ABB RobotStudio station: Universo_updated.rspag

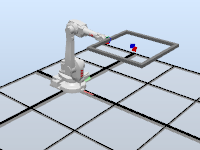
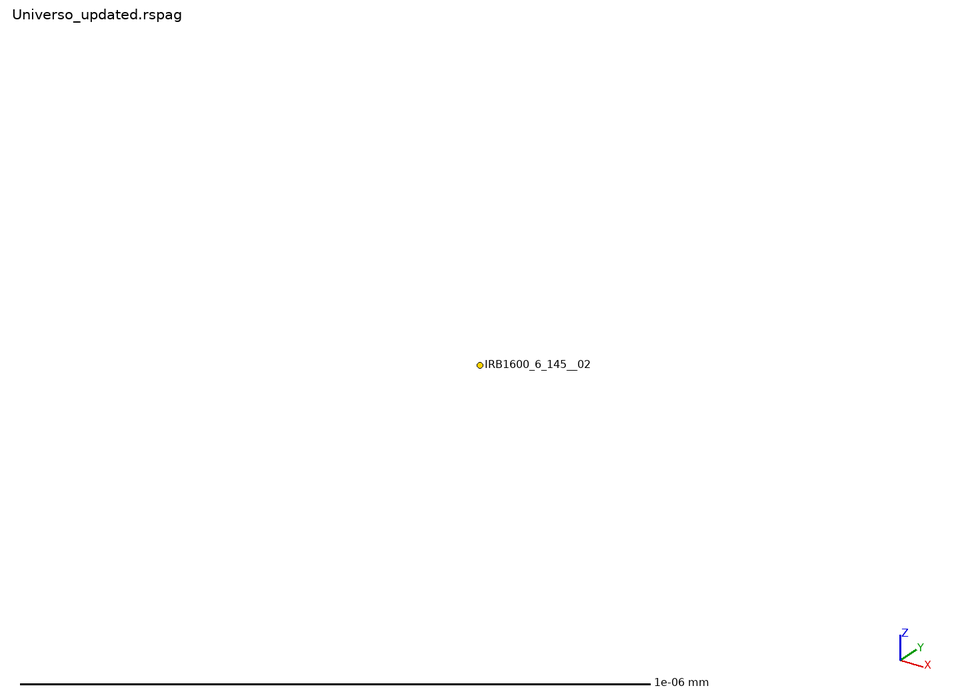
[picture v1: parts stored in the station drawn from their meshes, with robot base, taught points and paths (robot models come from the ABB library and are not in the file)]
--- station ---
Station Solution1 (saved by RobotStudio 22.1.9826.0)
Controller IRB1600_6_145
  mechanical unit ROB_1: IRB1600_6_145__02, 6 joints, base frame (0, 0, 0) mm
Layout (positions relative to the parent item):
  - IRB1600_6_145__02 [mechanism, from Robots\IRB1600_6_145_G_02.rslib] at (0, 0, 0) mm; joint values [-0.0012, -0.0048, 0.0813, -0.0158, -0.0765, 0.0158] (rad or m)
  - flange_connector [part, from Tools\IsoPlate_small_Binzel.rslib] at (809.87, -0.9, 1140.62) mm, rotated rx 0 ry 90 rz 0 deg
  - plane [part] at (1319.2, 1.57, 1145.26) mm, rotated rx 180 ry 0 rz 180 deg, size 1000 x 1000 x 50 mm
  - Frame_1 [frame]
  - Frame_2 [frame] at (-23.65, -1.83, 250.36) mm
Attachment: flange_connector is attached to IRB1600_6_145__02 / Link6
Attachment: plane is attached to flange_connector
Attachment: Workobject_2 is attached to IRB1600_6_145__02 / Link1
Targets, tools, work objects and paths stored in the station and not in the controller backup, written as RAPID:
! task T_ROB1
MODULE Module1
  LOCAL PERS wobjdata egm_wobj:=[FALSE,TRUE,"",[[0,0,0],[1,0,0,0]],[[0,0,0],[1,0,0,0]]];
  PROC EGM_CARTESIAN_MOVE()
    WaitTime 2;
  ENDPROC
ENDMODULE


--- Backups/IRB1600_6_145/RAPID/TASK1/PROGMOD/CalibData.mod ---
MODULE CalibData
    TASK PERS tooldata Tooldata_3:=[TRUE,[[-23.481,11.123,47.179],[0.707106781,0,0.707106781,0]],[1,[0,0,1],[1,0,0,0],0,0,0]];
    TASK PERS tooldata Tooldata_8:=[TRUE,[[35.292999999,18.761,1471.373000001],[0.707106781,0,-0.707106781,0]],[1,[0,0,1],[1,0,0,0],0,0,0]];
    TASK PERS tooldata Tooldata_4:=[TRUE,[[0,0,0],[1,0,0,0]],[1,[0,0,1],[1,0,0,0],0,0,0]];
    TASK PERS tooldata Tooldata_5:=[TRUE,[[0,0,0],[1,0,0,0]],[1,[0,0,1],[1,0,0,0],0,0,0]];
    TASK PERS tooldata Tooldata_6:=[TRUE,[[0,0,0],[1,0,0,0]],[1,[0,0,1],[1,0,0,0],0,0,0]];
    TASK PERS tooldata Tooldata_7:=[TRUE,[[-23.772999698,2.161000196,740.120999999],[0.707106781,0,-0.707106781,0]],[1,[0,0,1],[1,0,0,0],0,0,0]];
    TASK PERS wobjdata Workobject_2:=[FALSE,TRUE,"ROB_1",[[-55.133477186,-6.202200727,258.13059393],[1,0,0,0]],[[0,0,0],[1,0,0,0]]];
    TASK PERS tooldata Tooldata_9:=[TRUE,[[20.616002648,0.899999913,497.265999882],[0.707106781,-0.000000002,-0.707106781,0]],[1,[0,0,1],[1,0,0,0],0,0,0]];
    TASK PERS wobjdata Wobj_joint1:=[TRUE,FALSE,"ROB_1",[[639.116,-613.962,-938.233],[1,0,0,0]],[[0,0,0],[1,0,0,0]]];
ENDMODULE

--- Backups/IRB1600_6_145/RAPID/TASK1/PROGMOD/Module1.mod ---
MODULE Module1

     VAR robtarget position;
     VAR robtarget starting_position;
     VAR jointtarget joints;
     VAR speeddata velocity;
    TASK PERS wobjdata wobj:=[FALSE,FALSE,"ROB_1",[[639.116,-22.796,-980.437],[1,0,0,0]],[[0,0,0],[1,0,0,0]]];

    PROC main()

starting_position := CRobT(\TaskName:="T_ROB1" \Tool:=Tooldata_9 \WObj:=Workobject_2);
move 223,-627.8,7,20.4,0,0.9;
move 222,-628.9,7,20.4,15,1;
move 222,-630.1,6.9,20.4,15,1;
move 221,-631.2,6.9,20,15,1;
move 220,-632.5,6.9,20,15,1.1;
move 219,-633.7,6.8,19.6,15,1.1;
move 218,-635,6.8,19.6,15,1.2;
move 217,-636.4,6.8,19.2,15,1.2;
move 216,-637.8,6.8,19.2,15,1.2;
move 214,-639.3,6.8,18.8,15,1.3;
move 213,-640.8,6.8,18.8,15,1.3;
move 211,-642.4,6.8,18.4,14.9,1.4;
move 210,-644,6.8,18.4,14.9,1.4;
move 208,-645.6,6.7,18,14.9,1.5;
move 207,-647.3,6.7,18,14.9,1.5;
move 205,-649,6.7,17.6,14.9,1.6;
move 204,-650.7,6.7,17.6,14.9,1.6;
move 202,-652.4,6.6,17.2,14.9,1.7;
move 201,-654.1,6.6,16.8,14.8,1.7;
move 199,-655.8,6.6,16.8,14.8,1.8;
move 198,-657.5,6.6,16.8,14.8,1.9;
move 196,-659.2,6.6,16.4,14.8,1.9;
move 194,-660.8,6.6,16.4,14.8,2;
move 193,-662.4,6.6,16,14.7,2;
move 191,-664,6.6,15.6,14.7,2.1;
move 190,-665.6,6.5,15.6,14.7,2.2;
move 188,-667.2,6.5,15.2,14.7,2.2;
move 186,-668.7,6.5,15.2,14.6,2.3;
move 185,-670.2,6.5,14.8,14.6,2.4;
move 183,-671.6,6.5,14.8,14.6,2.4;
move 181,-673,6.5,14.4,14.5,2.5;
move 179,-674.3,6.5,14,14.5,2.6;
move 177,-675.5,6.4,14,14.5,2.7;
move 176,-676.7,6.4,13.6,14.5,2.7;
move 174,-677.8,6.4,13.2,14.4,2.8;
move 172,-678.8,6.4,13.2,14.4,2.9;
move 170,-679.8,6.4,12.8,14.3,2.9;
move 169,-680.7,6.4,12.8,14.3,3;
move 167,-681.6,6.4,12.4,14.3,3.1;
move 165,-682.4,6.4,12.4,14.2,3.2;
move 164,-683.2,6.4,12,14.2,3.3;
move 162,-683.9,6.4,11.6,14.2,3.3;
move 160,-684.7,6.3,11.6,14.1,3.4;
move 159,-685.4,6.3,11.2,14.1,3.5;
move 157,-686.1,6.3,11.2,14,3.6;
move 155,-686.7,6.3,10.8,14,3.6;
move 154,-687.4,6.3,10.8,13.9,3.7;
move 152,-688.1,6.3,10.4,13.9,3.8;
move 150,-688.8,6.2,10,13.8,3.9;
move 149,-689.5,6.2,10,13.8,4;
move 147,-690.2,6.2,9.6,13.7,4;
move 145,-690.9,6.2,9.6,13.7,4.1;
move 144,-691.6,6.2,9.2,13.6,4.2;
move 142,-692.3,6.2,9.2,13.6,4.3;
move 141,-693,6.1,8.8,13.5,4.3;
move 139,-693.6,6.1,8.8,13.5,4.4;
move 138,-694.3,6.1,8.4,13.4,4.5;
move 136,-694.9,6.1,8.4,13.4,4.6;
move 135,-695.5,6,8,13.3,4.6;
move 134,-696.1,6,8,13.3,4.7;
move 132,-696.6,6,7.6,13.2,4.8;
move 131,-697.1,5.9,7.6,13.1,4.9;
move 129,-697.6,5.9,7.2,13.1,4.9;
move 128,-698,5.9,7.2,13,5;
move 126,-698.4,5.8,6.8,12.9,5.1;
move 125,-698.8,5.8,6.8,12.9,5.1;
move 123,-699.2,5.8,6.4,12.8,5.2;
move 122,-699.5,5.7,6.4,12.8,5.3;
move 121,-699.8,5.7,6,12.7,5.4;
move 119,-700.1,5.6,6,12.6,5.4;
move 118,-700.3,5.6,5.6,12.6,5.5;
move 117,-700.6,5.6,5.6,12.5,5.6;
move 116,-700.8,5.5,5.6,12.4,5.6;
move 114,-701.1,5.5,5.2,12.3,5.7;
move 113,-701.3,5.4,5.2,12.3,5.8;
move 112,-701.6,5.4,4.8,12.2,5.8;
move 111,-701.8,5.3,4.8,12.1,5.9;
move 110,-702.1,5.2,4.8,12.1,6;
move 109,-702.4,5.2,4.4,12,6;
move 108,-702.7,5.1,4.4,11.9,6.1;
move 106,-703,5.1,4.4,11.8,6.2;
move 105,-703.3,5,4,11.7,6.2;
move 104,-703.7,4.9,4,11.7,6.3;
move 103,-704,4.9,3.6,11.6,6.3;
move 102,-704.4,4.8,3.6,11.5,6.4;
move 101,-704.8,4.7,3.6,11.4,6.5;
move 100,-705.2,4.7,3.2,11.3,6.5;
move 99,-705.6,4.6,3.2,11.3,6.6;
move 98,-706,4.5,3.2,11.2,6.7;
move 97,-706.4,4.5,2.8,11.1,6.7;
move 97,-706.8,4.4,2.8,11,6.8;
move 96,-707.2,4.3,2.8,10.9,6.8;
move 95,-707.6,4.3,2.8,10.8,6.9;
move 94,-708,4.2,2.4,10.8,7;
move 93,-708.4,4.1,2.4,10.7,7;
move 93,-708.7,4.1,2.4,10.6,7.1;
move 92,-709,4,2.4,10.5,7.1;
move 91,-709.3,3.9,2,10.4,7.2;
move 90,-709.6,3.9,2,10.3,7.2;
move 90,-709.8,3.8,2,10.2,7.3;
move 89,-710.1,3.7,2,10.1,7.4;
move 88,-710.3,3.6,1.6,10,7.4;
move 87,-710.5,3.6,1.6,9.9,7.5;
move 87,-710.6,3.5,1.6,9.8,7.5;
move 86,-710.8,3.5,1.6,9.8,7.6;
move 85,-710.9,3.4,1.2,9.7,7.6;
move 84,-711,3.3,1.2,9.6,7.7;
move 83,-711.1,3.3,1.2,9.5,7.7;
move 83,-711.2,3.2,0.8,9.4,7.8;
move 82,-711.2,3.1,0.8,9.3,7.8;
move 81,-711.3,3.1,0.8,9.2,7.9;
move 80,-711.4,3,0.8,9.1,7.9;
move 80,-711.4,3,0.4,9,8;
move 79,-711.4,2.9,0.4,8.9,8;
move 78,-711.5,2.9,0.4,8.8,8.1;
move 78,-711.4,2.8,0.4,8.7,8.1;
move 77,-711.4,2.8,0.4,8.6,8.2;
move 77,-711.4,2.7,0,8.5,8.2;
move 76,-711.4,2.7,0,8.4,8.3;
move 75,-711.4,2.6,0,8.3,8.3;
move 75,-711.4,2.6,-0,8.2,8.4;
move 74,-711.4,2.5,-0,8,8.4;
move 73,-711.3,2.5,-0.4,7.9,8.4;
move 73,-711.3,2.5,-0.4,7.8,8.5;
move 72,-711.2,2.4,-0.4,7.7,8.5;
move 71,-711.2,2.4,-0.4,7.6,8.6;
move 70,-711.1,2.4,-0.8,7.5,8.6;
move 69,-711.1,2.3,-0.8,7.4,8.7;
move 69,-711,2.3,-0.8,7.3,8.7;
move 68,-711,2.2,-1.2,7.2,8.7;
move 67,-710.9,2.2,-1.2,7.1,8.8;
move 66,-710.9,2.2,-1.2,7,8.8;
move 66,-710.9,2.1,-1.2,6.9,8.8;
move 65,-710.8,2.1,-1.6,6.7,8.9;
move 64,-710.8,2.1,-1.6,6.6,8.9;
move 64,-710.8,2,-1.6,6.5,9;
move 63,-710.7,2,-1.6,6.4,9;
move 62,-710.7,2,-1.6,6.3,9;
move 61,-710.6,2,-2,6.2,9.1;
move 61,-710.6,2,-2,6.1,9.1;
move 60,-710.5,2,-2,6,9.1;
move 59,-710.5,2,-2.4,5.8,9.2;
move 59,-710.4,2,-2.4,5.7,9.2;
move 58,-710.3,2,-2.4,5.6,9.2;
move 58,-710.2,2,-2.4,5.5,9.3;
move 57,-710.1,2,-2.4,5.4,9.3;
move 56,-710,2,-2.4,5.3,9.3;
move 56,-709.8,2,-2.8,5.1,9.4;
move 55,-709.7,2,-2.8,5,9.4;
move 54,-709.5,2,-2.8,4.9,9.4;
move 54,-709.3,2,-2.8,4.8,9.5;
move 53,-709.1,2.1,-3.2,4.7,9.5;
move 53,-708.8,2.1,-3.2,4.5,9.5;
move 52,-708.5,2.1,-3.2,4.4,9.5;
move 52,-708.3,2.1,-3.2,4.3,9.6;
move 51,-707.9,2.1,-3.2,4.2,9.6;
move 51,-707.6,2.1,-3.2,4.1,9.6;
move 50,-707.3,2.1,-3.6,3.9,9.7;
move 50,-706.9,2.1,-3.6,3.8,9.7;
move 49,-706.5,2.2,-3.6,3.7,9.7;
move 49,-706.1,2.2,-3.6,3.6,9.7;
move 48,-705.6,2.2,-3.6,3.5,9.7;
move 48,-705.2,2.2,-3.6,3.3,9.8;
move 47,-704.7,2.3,-4,3.2,9.8;
move 47,-704.3,2.3,-4,3.1,9.8;
move 47,-703.8,2.3,-4,3,9.8;
move 47,-703.4,2.3,-4,2.9,9.8;
move 46,-702.9,2.4,-4,2.7,9.9;
move 46,-702.4,2.4,-4,2.6,9.9;
move 46,-701.9,2.4,-4,2.5,9.9;
move 46,-701.4,2.4,-4,2.4,9.9;
move 46,-700.9,2.4,-4,2.2,9.9;
move 46,-700.3,2.5,-4,2.1,9.9;
move 46,-699.8,2.5,-4,2,9.9;
move 46,-699.3,2.5,-4,1.9,9.9;
move 46,-698.7,2.5,-4,1.7,9.9;
move 46,-698.1,2.5,-4,1.6,9.9;
move 46,-697.5,2.6,-4,1.5,10;
move 47,-696.9,2.6,-4,1.4,10;
move 47,-696.3,2.6,-4,1.2,10;
move 47,-695.7,2.7,-4,1.1,10;
move 48,-695.1,2.7,-3.6,1,10;
move 48,-694.5,2.7,-3.6,0.9,10;
move 48,-693.8,2.7,-3.6,0.7,10;
move 49,-693.2,2.7,-3.6,0.6,10;
move 49,-692.6,2.7,-3.6,0.5,10;
move 50,-692,2.7,-3.6,0.4,10;
move 50,-691.5,2.7,-3.6,0.2,10;
move 51,-690.9,2.7,-3.2,0.1,10;
move 52,-690.4,2.8,-3.2,-0,10;
move 52,-689.8,2.8,-3.2,-0.1,10;
move 53,-689.3,2.8,-3.2,-0.3,10;
move 54,-688.7,2.8,-2.8,-0.4,10;
move 55,-688.2,2.8,-2.8,-0.5,10;
move 56,-687.7,2.8,-2.8,-0.6,10;
move 56,-687.2,2.8,-2.4,-0.8,10;
move 57,-686.7,2.8,-2.4,-0.9,10;
move 58,-686.3,2.8,-2.4,-1,10;
move 59,-685.9,2.8,-2.4,-1.1,10;
move 60,-685.4,2.8,-2,-1.3,10;
move 61,-685,2.8,-2,-1.4,10;
move 62,-684.6,2.8,-2,-1.5,10;
move 63,-684.3,2.8,-1.6,-1.6,9.9;
move 64,-683.9,2.9,-1.6,-1.8,9.9;
move 65,-683.6,2.9,-1.6,-1.9,9.9;
move 66,-683.3,2.9,-1.2,-2,9.9;
move 66,-683,2.9,-1.2,-2.1,9.9;
move 67,-682.8,2.9,-1.2,-2.3,9.9;
move 68,-682.6,2.9,-0.8,-2.4,9.9;
move 69,-682.5,2.9,-0.8,-2.5,9.9;
move 70,-682.4,2.9,-0.8,-2.6,9.9;
move 71,-682.3,2.9,-0.4,-2.7,9.8;
move 72,-682.2,2.9,-0.4,-2.9,9.8;
move 73,-682.2,2.9,-0.4,-3,9.8;
move 74,-682.3,2.9,-0,-3.1,9.8;
move 75,-682.3,2.9,-0,-3.2,9.8;
move 76,-682.4,3,0,-3.4,9.7;
move 77,-682.5,3,0.4,-3.5,9.7;
move 78,-682.6,3,0.4,-3.6,9.7;
move 79,-682.8,2.9,0.4,-3.7,9.7;
move 80,-683,2.9,0.8,-3.8,9.7;
move 81,-683.2,2.9,0.8,-4,9.6;
move 81,-683.5,2.9,0.8,-4.1,9.6;
move 82,-683.7,2.9,0.8,-4.2,9.6;
move 83,-684,2.9,1.2,-4.3,9.5;
move 84,-684.2,2.9,1.2,-4.4,9.5;
move 84,-684.5,2.9,1.2,-4.6,9.5;
move 85,-684.8,2.9,1.2,-4.7,9.5;
move 85,-685.1,2.9,1.6,-4.8,9.4;
move 86,-685.5,2.9,1.6,-4.9,9.4;
move 86,-685.9,2.9,1.6,-5,9.4;
move 86,-686.2,2.9,1.6,-5.2,9.3;
move 87,-686.6,2.9,1.6,-5.3,9.3;
move 87,-687.1,2.9,1.6,-5.4,9.3;
move 87,-687.5,2.9,1.6,-5.5,9.2;
move 86,-688,2.8,1.6,-5.6,9.2;
move 86,-688.6,2.8,1.6,-5.7,9.2;
move 86,-689.1,2.8,1.6,-5.9,9.1;
move 85,-689.7,2.8,1.6,-6,9.1;
move 84,-690.4,2.7,1.2,-6.1,9;
move 84,-691.1,2.7,1.2,-6.2,9;
move 83,-691.8,2.7,1.2,-6.3,9;
move 82,-692.5,2.6,0.8,-6.4,8.9;
move 81,-693.3,2.6,0.8,-6.5,8.9;
move 80,-694.1,2.6,0.8,-6.6,8.9;
move 79,-694.9,2.5,0.4,-6.8,8.8;
move 78,-695.8,2.5,0.4,-6.9,8.8;
move 77,-696.7,2.4,0.4,-7,8.7;
move 75,-697.6,2.4,-0,-7.1,8.7;
move 74,-698.5,2.3,-0,-7.2,8.7;
move 72,-699.4,2.3,-0.4,-7.3,8.6;
move 71,-700.2,2.2,-0.4,-7.4,8.6;
move 69,-701.1,2.1,-0.8,-7.5,8.5;
move 67,-701.9,2,-1.2,-7.6,8.5;
move 65,-702.7,2,-1.2,-7.7,8.5;
move 64,-703.4,1.9,-1.6,-7.8,8.4;
move 62,-704.1,1.8,-2,-8,8.4;
move 60,-704.8,1.7,-2,-8.1,8.3;
move 58,-705.3,1.6,-2.4,-8.2,8.3;
move 56,-705.9,1.5,-2.8,-8.3,8.2;
move 54,-706.3,1.4,-2.8,-8.4,8.2;
move 51,-706.7,1.3,-3.2,-8.5,8.2;
move 49,-707,1.2,-3.6,-8.6,8.1;
move 47,-707.2,1.1,-3.6,-8.7,8.1;
move 45,-707.3,1,-4,-8.8,8;
move 42,-707.3,0.9,-4.4,-8.9,8;
move 40,-707.2,0.8,-4.8,-9,7.9;
move 37,-707.1,0.7,-5.2,-9.1,7.9;
move 35,-706.8,0.6,-5.6,-9.2,7.8;
move 32,-706.5,0.4,-6,-9.3,7.8;
move 29,-706.1,0.3,-6.4,-9.4,7.7;
move 27,-705.6,0.2,-6.8,-9.5,7.7;
move 24,-705,0.1,-6.8,-9.6,7.6;
move 22,-704.3,-0.1,-7.2,-9.7,7.6;
move 19,-703.5,-0.2,-7.6,-9.8,7.5;
move 16,-702.7,-0.4,-8,-9.9,7.4;
move 13,-701.9,-0.5,-8.4,-10,7.4;
move 11,-701,-0.7,-8.8,-10,7.3;
move 8,-700.1,-0.8,-9.2,-10.1,7.3;
move 5,-699.1,-1,-9.6,-10.2,7.2;
move 2,-698.1,-1.1,-10,-10.3,7.2;
move -1,-697.1,-1.3,-10.4,-10.4,7.1;
move -3,-696.2,-1.4,-10.8,-10.5,7.1;
move -6,-695.2,-1.6,-11.2,-10.6,7;
move -9,-694.2,-1.7,-11.6,-10.7,6.9;
move -11,-693.2,-1.9,-12,-10.8,6.9;
move -14,-692.1,-2.1,-12,-10.9,6.8;
move -16,-691.1,-2.2,-12.4,-10.9,6.8;
move -18,-690.1,-2.4,-12.8,-11,6.7;
move -21,-689,-2.5,-13.2,-11.1,6.6;
move -23,-688,-2.7,-13.2,-11.2,6.6;
move -25,-686.9,-2.8,-13.6,-11.3,6.5;
move -27,-685.7,-3,-14,-11.4,6.4;
move -29,-684.5,-3.1,-14.4,-11.4,6.4;
move -31,-683.1,-3.3,-14.8,-11.5,6.3;
move -33,-681.7,-3.4,-14.8,-11.6,6.3;
move -35,-680.1,-3.6,-15.2,-11.7,6.2;
move -37,-678.5,-3.7,-15.6,-11.8,6.1;
move -38,-676.6,-3.8,-15.6,-11.8,6.1;
move -40,-674.7,-4,-15.6,-11.9,6;
move -41,-672.5,-4.1,-16,-12,5.9;
move -42,-670.2,-4.2,-16,-12.1,5.9;
move -44,-667.7,-4.4,-16.4,-12.1,5.8;
move -45,-665,-4.5,-16.4,-12.2,5.7;
move -45,-662.1,-4.6,-16.4,-12.3,5.7;
move -46,-659,-4.7,-16.8,-12.4,5.6;
move -47,-655.8,-4.8,-16.8,-12.4,5.5;
move -47,-652.4,-4.9,-16.8,-12.5,5.5;
move -48,-648.9,-5.1,-16.8,-12.6,5.4;
move -48,-645.3,-5.2,-16.8,-12.6,5.3;
move -48,-641.6,-5.3,-17.2,-12.7,5.2;
move -49,-637.9,-5.3,-17.2,-12.8,5.2;
move -49,-634.1,-5.4,-16.8,-12.8,5.1;
move -49,-630.3,-5.5,-16.8,-12.9,5;
move -48,-626.6,-5.6,-16.8,-13,5;
move -48,-622.9,-5.7,-16.8,-13,4.9;
move -48,-619.3,-5.8,-16.8,-13.1,4.8;
move -48,-615.8,-5.8,-16.8,-13.1,4.7;
move -47,-612.5,-5.9,-16.8,-13.2,4.7;
move -47,-609.3,-6,-16.8,-13.3,4.6;
move -46,-606.3,-6,-16.8,-13.3,4.5;
move -46,-603.6,-6.1,-16.4,-13.4,4.4;
move -45,-601,-6.1,-16.4,-13.4,4.4;
move -44,-598.7,-6.2,-16.4,-13.5,4.3;
move -43,-596.6,-6.2,-16,-13.5,4.2;
move -42,-594.8,-6.3,-16,-13.6,4.1;
move -41,-593.2,-6.3,-16,-13.6,4.1;
move -40,-591.9,-6.4,-15.6,-13.7,4;
move -39,-590.7,-6.4,-15.6,-13.7,3.9;
move -38,-589.8,-6.5,-15.6,-13.8,3.8;
move -37,-589.2,-6.5,-15.2,-13.8,3.8;
move -35,-588.7,-6.5,-15.2,-13.9,3.7;
move -34,-588.4,-6.6,-14.8,-13.9,3.6;
move -32,-588.2,-6.6,-14.8,-14,3.5;
move -31,-588.2,-6.6,-14.4,-14,3.5;
move -29,-588.3,-6.7,-14.4,-14.1,3.4;
move -27,-588.5,-6.7,-14,-14.1,3.3;
move -26,-588.8,-6.7,-13.6,-14.2,3.2;
move -24,-589.1,-6.7,-13.6,-14.2,3.1;
move -22,-589.4,-6.8,-13.2,-14.2,3.1;
move -21,-589.7,-6.8,-13.2,-14.3,3;
move -19,-589.9,-6.8,-12.8,-14.3,2.9;
move -17,-590.2,-6.9,-12.4,-14.4,2.8;
move -15,-590.3,-6.9,-12.4,-14.4,2.7;
move -14,-590.4,-6.9,-12,-14.4,2.7;
move -12,-590.4,-7,-12,-14.5,2.6;
move -10,-590.3,-7,-11.6,-14.5,2.5;
move -9,-590,-7,-11.6,-14.5,2.4;
move -7,-589.7,-7,-11.2,-14.6,2.3;
move -5,-589.2,-7.1,-10.8,-14.6,2.3;
move -3,-588.6,-7.1,-10.8,-14.6,2.2;
move -1,-588,-7.1,-10.4,-14.6,2.1;
move 1,-587.2,-7.2,-10,-14.7,2;
move 3,-586.3,-7.2,-10,-14.7,1.9;
move 5,-585.4,-7.2,-9.6,-14.7,1.9;
move 7,-584.3,-7.3,-9.2,-14.7,1.8;
move 9,-583.2,-7.3,-9.2,-14.8,1.7;
move 10,-582.1,-7.4,-8.8,-14.8,1.6;
move 12,-580.9,-7.4,-8.4,-14.8,1.5;
move 14,-579.6,-7.5,-8.4,-14.8,1.5;
move 16,-578.3,-7.5,-8,-14.8,1.4;
move 18,-577,-7.5,-7.6,-14.9,1.3;
move 20,-575.6,-7.6,-7.6,-14.9,1.2;
move 22,-574.3,-7.6,-7.2,-14.9,1.1;
move 24,-573,-7.7,-7.2,-14.9,1;
move 26,-571.7,-7.7,-6.8,-14.9,1;
move 28,-570.4,-7.7,-6.4,-14.9,0.9;
move 30,-569.2,-7.8,-6.4,-14.9,0.8;
move 32,-568,-7.8,-6,-15,0.7;
move 34,-566.8,-7.8,-5.6,-15,0.6;
move 36,-565.6,-7.9,-5.2,-15,0.5;
move 38,-564.5,-7.9,-5.2,-15,0.5;
move 40,-563.5,-8,-4.8,-15,0.4;
move 42,-562.5,-8,-4.8,-15,0.3;
move 44,-561.5,-8,-4.4,-15,0.2;
move 46,-560.7,-8.1,-4,-15,0.1;
move 48,-559.8,-8.1,-3.6,-15,0;
move 50,-559.1,-8.1,-3.6,-15,-0;
move 52,-558.3,-8.2,-3.2,-15,-0.1;
move 54,-557.7,-8.2,-2.8,-15,-0.2;
move 57,-557.1,-8.2,-2.4,-15,-0.3;
move 59,-556.5,-8.2,-2.4,-15,-0.4;
move 61,-556.1,-8.2,-2,-15,-0.4;
move 63,-555.6,-8.2,-1.6,-15,-0.5;
move 66,-555.2,-8.2,-1.2,-15,-0.6;
move 68,-554.9,-8.2,-1.2,-15,-0.7;
move 70,-554.6,-8.2,-0.8,-15,-0.8;
move 72,-554.3,-8.3,-0.4,-15,-0.9;
move 75,-554.1,-8.3,-0,-14.9,-0.9;
move 77,-554,-8.3,0.4,-14.9,-1;
move 79,-553.8,-8.3,0.8,-14.9,-1.1;
move 81,-553.8,-8.3,0.8,-14.9,-1.2;
move 83,-553.8,-8.3,1.2,-14.9,-1.3;
move 86,-553.8,-8.2,1.2,-14.9,-1.3;
move 88,-553.9,-8.2,1.6,-14.9,-1.4;
move 90,-554.1,-8.2,2,-14.8,-1.5;
move 92,-554.3,-8.2,2.4,-14.8,-1.6;
move 94,-554.6,-8.1,2.4,-14.8,-1.7;
move 96,-555,-8.1,2.8,-14.8,-1.8;
move 98,-555.4,-8.1,3.2,-14.8,-1.8;
move 100,-555.9,-8,3.6,-14.7,-1.9;
move 102,-556.4,-8,3.6,-14.7,-2;
move 104,-557.1,-8,4,-14.7,-2.1;
move 106,-557.8,-7.9,4.4,-14.7,-2.2;
move 107,-558.6,-7.8,4.4,-14.6,-2.2;
move 109,-559.5,-7.7,4.8,-14.6,-2.3;
move 111,-560.5,-7.7,4.8,-14.6,-2.4;
move 112,-561.5,-7.6,5.2,-14.5,-2.5;
move 113,-562.7,-7.5,5.2,-14.5,-2.6;
move 115,-563.9,-7.4,5.2,-14.5,-2.6;
move 116,-565.3,-7.4,5.6,-14.4,-2.7;
move 117,-566.6,-7.3,5.6,-14.4,-2.8;
move 118,-568.1,-7.2,6,-14.4,-2.9;
move 120,-569.5,-7.2,6,-14.3,-3;
move 121,-571.1,-7.1,6.4,-14.3,-3;
move 122,-572.6,-7,6.4,-14.3,-3.1;
move 123,-574.2,-6.9,6.4,-14.2,-3.2;
move 124,-575.8,-6.8,6.8,-14.2,-3.3;
move 125,-577.5,-6.7,6.8,-14.1,-3.3;
move 126,-579.1,-6.6,6.8,-14.1,-3.4;
move 126,-580.8,-6.4,6.8,-14.1,-3.5;
move 127,-582.4,-6.3,7.2,-14,-3.6;
move 128,-584,-6.2,7.2,-14,-3.7;
move 129,-585.6,-6.1,7.2,-13.9,-3.7;
move 130,-587.1,-5.9,7.2,-13.9,-3.8;
move 130,-588.5,-5.8,7.6,-13.8,-3.9;
move 131,-589.9,-5.7,7.6,-13.8,-4;
move 132,-591.3,-5.6,7.6,-13.7,-4;
move 132,-592.6,-5.4,8,-13.7,-4.1;
move 133,-593.8,-5.3,8,-13.6,-4.2;
move 133,-594.9,-5.2,8,-13.6,-4.3;
move 134,-596,-5.1,8,-13.5,-4.3;
move 134,-596.9,-4.9,8,-13.5,-4.4;
move 134,-597.7,-4.8,8,-13.4,-4.5;
move 135,-598.4,-4.7,8,-13.4,-4.6;
move 135,-599,-4.6,8,-13.3,-4.6;
move 135,-599.6,-4.5,8,-13.2,-4.7;
move 135,-599.9,-4.3,8,-13.2,-4.8;
move 136,-600.2,-4.2,8.4,-13.1,-4.9;
move 136,-600.5,-4.1,8.4,-13.1,-4.9;
move 136,-600.7,-4,8.4,-13,-5;
move 137,-600.9,-3.9,8.4,-12.9,-5.1;
move 137,-601,-3.8,8.4,-12.9,-5.1;
move 137,-600.9,-3.7,8.4,-12.8,-5.2;
move 137,-600.7,-3.6,8.4,-12.7,-5.3;
move 137,-600.4,-3.5,8.4,-12.7,-5.4;
move 137,-600.1,-3.3,8.4,-12.6,-5.4;
move 137,-599.7,-3.2,8.4,-12.5,-5.5;
move 137,-599.4,-3.1,8.4,-12.5,-5.6;
move 137,-599,-3,8.4,-12.4,-5.6;
move 137,-598.6,-2.9,8.4,-12.3,-5.7;
move 137,-598.2,-2.8,8.4,-12.3,-5.8;
move 137,-597.9,-2.7,8.4,-12.2,-5.8;
move 137,-597.6,-2.6,8.4,-12.1,-5.9;
move 137,-597.4,-2.5,8.4,-12,-6;
move 137,-597.1,-2.4,8.4,-12,-6;
move 137,-597,-2.3,8.4,-11.9,-6.1;
move 137,-596.8,-2.3,8.4,-11.8,-6.2;
move 137,-596.8,-2.2,8.4,-11.7,-6.2;
move 137,-596.9,-2.1,8.4,-11.7,-6.3;
move 137,-597,-2,8.4,-11.6,-6.3;
move 137,-597.3,-2,8.4,-11.5,-6.4;
move 137,-597.6,-1.9,8.4,-11.4,-6.5;
move 137,-598.1,-1.8,8.4,-11.3,-6.5;
move 137,-598.7,-1.7,8.4,-11.3,-6.6;
move 137,-599.5,-1.7,8.4,-11.2,-6.7;
move 137,-600.3,-1.6,8.4,-11.1,-6.7;
move 137,-601.3,-1.6,8.4,-11,-6.8;
move 137,-602.4,-1.5,8.4,-10.9,-6.8;
move 137,-603.6,-1.5,8.4,-10.8,-6.9;
move 137,-604.9,-1.4,8.4,-10.7,-7;
move 137,-606.3,-1.3,8.4,-10.7,-7;
move 137,-607.8,-1.3,8.4,-10.6,-7.1;
move 136,-609.3,-1.2,8.4,-10.5,-7.1;
move 136,-610.9,-1.1,8.4,-10.4,-7.2;
move 136,-612.5,-1.1,8.4,-10.3,-7.2;
move 135,-614.2,-1,8,-10.2,-7.3;
move 135,-615.8,-1,8,-10.1,-7.4;
move 134,-617.5,-0.9,8,-10,-7.4;
move 134,-619.1,-0.9,8,-9.9,-7.5;
move 133,-620.7,-0.8,8,-9.8,-7.5;
move 132,-622.3,-0.7,8,-9.7,-7.6;
move 132,-623.8,-0.7,7.6,-9.6,-7.6;
move 131,-625.2,-0.6,7.6,-9.6,-7.7;
move 130,-626.6,-0.6,7.6,-9.5,-7.7;
move 129,-627.9,-0.5,7.2,-9.4,-7.8;
move 128,-629.2,-0.5,7.2,-9.3,-7.8;
move 127,-630.4,-0.4,7.2,-9.2,-7.9;
move 126,-631.5,-0.3,6.8,-9.1,-7.9;
move 124,-632.6,-0.3,6.8,-9,-8;
move 123,-633.5,-0.2,6.4,-8.9,-8;
move 122,-634.4,-0.1,6.4,-8.8,-8.1;
move 120,-635.4,-0.1,6,-8.7,-8.1;
move 119,-636.4,-0,6,-8.6,-8.2;
move 117,-637.4,0.1,5.6,-8.5,-8.2;
move 116,-638.3,0.1,5.6,-8.3,-8.3;
move 114,-639.3,0.2,5.2,-8.2,-8.3;
move 113,-640.1,0.2,5.2,-8.1,-8.4;
move 111,-641,0.3,4.8,-8,-8.4;
move 109,-641.7,0.4,4.8,-7.9,-8.4;
move 107,-642.4,0.5,4.4,-7.8,-8.5;
move 105,-643.1,0.5,4,-7.7,-8.5;
move 104,-643.8,0.6,4,-7.6,-8.6;
move 102,-644.4,0.7,3.6,-7.5,-8.6;
move 100,-645,0.8,3.2,-7.4,-8.7;
move 98,-645.5,0.9,3.2,-7.3,-8.7;
move 96,-646,0.9,2.8,-7.2,-8.7;
move 94,-646.4,1,2.4,-7.1,-8.8;
move 91,-646.7,1.1,2,-7,-8.8;
move 89,-647,1.2,2,-6.8,-8.8;
move 87,-647.1,1.3,1.6,-6.7,-8.9;
move 85,-647.2,1.4,1.2,-6.6,-8.9;
move 83,-647.2,1.5,1.2,-6.5,-9;
move 81,-647.1,1.5,0.8,-6.4,-9;
move 79,-646.9,1.6,0.4,-6.3,-9;
move 77,-646.6,1.7,0.4,-6.2,-9.1;
move 75,-646.3,1.8,-0,-6,-9.1;
move 72,-645.9,1.9,-0.4,-5.9,-9.1;
move 70,-645.4,1.9,-0.8,-5.8,-9.2;
move 68,-644.9,2,-1.2,-5.7,-9.2;
move 66,-644.3,2.1,-1.2,-5.6,-9.2;
move 64,-643.7,2.2,-1.6,-5.5,-9.3;
move 62,-643.1,2.3,-2,-5.4,-9.3;
move 59,-642.4,2.4,-2,-5.2,-9.3;
move 57,-641.7,2.5,-2.4,-5.1,-9.4;
move 55,-641,2.5,-2.8,-5,-9.4;
move 53,-640.3,2.6,-3.2,-4.9,-9.4;
move 51,-639.6,2.7,-3.2,-4.8,-9.5;
move 49,-638.9,2.8,-3.6,-4.6,-9.5;
move 46,-638.2,2.9,-4,-4.5,-9.5;
move 44,-637.6,2.9,-4.4,-4.4,-9.5;
move 42,-637,3,-4.4,-4.3,-9.6;
move 40,-636.4,3.1,-4.8,-4.2,-9.6;
move 37,-635.9,3.2,-5.2,-4.1,-9.6;
move 35,-635.4,3.3,-5.6,-3.9,-9.7;
move 33,-635,3.4,-5.6,-3.8,-9.7;
move 30,-634.5,3.5,-6,-3.7,-9.7;
move 28,-634.1,3.5,-6.4,-3.6,-9.7;
move 25,-633.7,3.6,-6.8,-3.4,-9.7;
move 23,-633.3,3.7,-7.2,-3.3,-9.8;
move 20,-632.9,3.8,-7.6,-3.2,-9.8;
move 18,-632.4,3.9,-8,-3.1,-9.8;
move 15,-632,4,-8,-3,-9.8;
move 13,-631.5,4,-8.4,-2.8,-9.8;
move 10,-631.1,4.1,-8.8,-2.7,-9.9;
move 8,-630.6,4.2,-9.2,-2.6,-9.9;
move 6,-630.1,4.3,-9.6,-2.5,-9.9;
move 3,-629.5,4.3,-10,-2.3,-9.9;
move 1,-628.9,4.4,-10.4,-2.2,-9.9;
move -1,-628.3,4.5,-10.4,-2.1,-9.9;
move -3,-627.7,4.6,-10.8,-2,-9.9;
move -5,-627.1,4.6,-11.2,-1.8,-9.9;
move -7,-626.4,4.7,-11.2,-1.7,-9.9;
move -9,-625.7,4.8,-11.6,-1.6,-9.9;
move -11,-624.9,4.9,-11.6,-1.5,-10;
move -13,-624.2,4.9,-12,-1.3,-10;
move -15,-623.4,5,-12.4,-1.2,-10;
move -16,-622.6,5.1,-12.4,-1.1,-10;
move -18,-621.7,5.2,-12.8,-1,-10;
move -20,-620.8,5.2,-12.8,-0.8,-10;
move -22,-619.8,5.3,-13.2,-0.7,-10;
move -23,-618.8,5.4,-13.6,-0.6,-10;
move -25,-617.7,5.4,-13.6,-0.5,-10;
move -27,-616.6,5.5,-14,-0.3,-10;
move -29,-615.5,5.5,-14,-0.2,-10;
move -30,-614.3,5.5,-14.4,-0.1,-10;
move -32,-613.1,5.6,-14.8,0,-10;
move -33,-611.8,5.6,-14.8,0.2,-10;
move -35,-610.4,5.7,-15.2,0.3,-10;
move -36,-609,5.7,-15.2,0.4,-10;
move -38,-607.5,5.7,-15.6,0.5,-10;
move -39,-606,5.8,-15.6,0.7,-10;
move -40,-604.4,5.8,-15.6,0.8,-10;
move -42,-602.8,5.8,-16,0.9,-10;
move -43,-601.2,5.8,-16,1,-10;
move -44,-599.5,5.9,-16.4,1.1,-10;
move -45,-597.8,5.9,-16.4,1.3,-10;
move -46,-596,5.9,-16.8,1.4,-10;
move -47,-594.3,6,-16.8,1.5,-10;
move -48,-592.4,6,-16.8,1.6,-9.9;
move -49,-590.6,6,-16.8,1.8,-9.9;
move -49,-588.8,6,-17.2,1.9,-9.9;
move -50,-586.9,6,-17.2,2,-9.9;
move -50,-585,6,-17.2,2.1,-9.9;
move -50,-583.1,6,-17.2,2.3,-9.9;
move -51,-581.3,6,-17.2,2.4,-9.9;
move -51,-579.4,6,-17.2,2.5,-9.9;
move -51,-577.5,6,-17.2,2.6,-9.9;
move -51,-575.7,6,-17.2,2.8,-9.8;
move -51,-573.8,6,-17.2,2.9,-9.8;
move -51,-572,6,-17.2,3,-9.8;
move -51,-570.1,6,-17.2,3.1,-9.8;
move -50,-568.1,6,-17.2,3.3,-9.8;
move -50,-566.2,6,-17.2,3.4,-9.7;
move -49,-564.2,6,-17.2,3.5,-9.7;
move -49,-562.2,5.9,-16.8,3.6,-9.7;
move -48,-560.1,5.9,-16.8,3.7,-9.7;
move -47,-557.9,5.9,-16.8,3.9,-9.7;
move -47,-555.7,5.9,-16.8,4,-9.6;
move -46,-553.3,5.9,-16.4,4.1,-9.6;
move -45,-550.9,5.9,-16.4,4.2,-9.6;
move -44,-548.4,5.9,-16.4,4.3,-9.5;
move -42,-545.8,5.9,-16,4.5,-9.5;
move -41,-543,5.9,-16,4.6,-9.5;
move -40,-540.2,5.9,-15.6,4.7,-9.5;
move -38,-537.3,5.9,-15.6,4.8,-9.4;
move -37,-534.3,5.8,-15.2,4.9,-9.4;
move -36,-531.3,5.8,-15.2,5.1,-9.4;
move -34,-528.1,5.9,-14.8,5.2,-9.3;
move -33,-525,5.8,-14.8,5.3,-9.3;
move -31,-521.8,5.8,-14.4,5.4,-9.3;
move -30,-518.7,5.8,-14.4,5.5,-9.2;
move -28,-515.6,5.8,-14,5.6,-9.2;
move -27,-512.6,5.8,-14,5.8,-9.2;
move -25,-509.6,5.8,-13.6,5.9,-9.1;
move -24,-506.8,5.8,-13.6,6,-9.1;
move -22,-504.2,5.8,-13.2,6.1,-9;
move -21,-501.7,5.8,-13.2,6.2,-9;
move -19,-499.5,5.9,-12.8,6.3,-9;
move -18,-497.5,5.9,-12.8,6.4,-8.9;
move -16,-495.7,5.9,-12.4,6.5,-8.9;
move -15,-494.2,5.9,-12.4,6.7,-8.9;
move -13,-492.8,5.9,-12,6.8,-8.8;
move -11,-491.8,5.9,-11.6,6.9,-8.8;
move -10,-490.9,5.9,-11.6,7,-8.7;
move -8,-490.3,5.9,-11.2,7.1,-8.7;
move -7,-489.9,5.9,-11.2,7.2,-8.7;
move -6,-489.6,5.9,-10.8,7.3,-8.6;
move -4,-489.5,6,-10.8,7.4,-8.6;
move -3,-489.6,6,-10.8,7.5,-8.5;
move -2,-489.8,6,-10.4,7.7,-8.5;
move -1,-490,6,-10.4,7.8,-8.5;
move 0,-490.3,6,-10,7.9,-8.4;
move 1,-490.7,6.1,-10,8,-8.4;
move 2,-491.1,6.1,-10,8.1,-8.3;
move 3,-491.5,6.1,-10,8.2,-8.3;
move 3,-491.9,6.2,-9.6,8.3,-8.2;
move 4,-492.3,6.2,-9.6,8.4,-8.2;
move 5,-492.7,6.3,-9.6,8.5,-8.1;
move 5,-493,6.3,-9.6,8.6,-8.1;
move 6,-493.3,6.3,-9.6,8.7,-8;
move 6,-493.5,6.4,-9.2,8.8,-8;
move 6,-493.7,6.4,-9.2,8.9,-7.9;
move 6,-493.8,6.4,-9.2,9,-7.9;
move 6,-493.8,6.5,-9.2,9.1,-7.8;
move 6,-493.8,6.5,-9.2,9.2,-7.8;
move 6,-493.8,6.6,-9.2,9.3,-7.7;
move 5,-493.7,6.6,-9.6,9.4,-7.7;
move 5,-493.6,6.6,-9.6,9.5,-7.6;
move 4,-493.4,6.7,-9.6,9.6,-7.6;
move 3,-493.1,6.7,-9.6,9.7,-7.5;
move 2,-492.8,6.8,-10,9.8,-7.5;
move 1,-492.5,6.8,-10,9.9,-7.4;
move 0,-492.1,6.8,-10,10,-7.4;
move -1,-491.8,6.9,-10.4,10.1,-7.3;
move -2,-491.4,6.9,-10.4,10.2,-7.3;
move -4,-491,7,-10.8,10.2,-7.2;
move -5,-490.6,7,-10.8,10.3,-7.1;
move -7,-490.1,7,-11.2,10.4,-7.1;
move -8,-489.7,7.1,-11.2,10.5,-7;
move -10,-489.2,7.1,-11.6,10.6,-7;
move -12,-488.7,7.2,-11.6,10.7,-6.9;
move -14,-488.1,7.3,-12,10.8,-6.8;
move -15,-487.6,7.3,-12.4,10.9,-6.8;
move -17,-487,7.4,-12.8,11,-6.7;
move -19,-486.3,7.5,-12.8,11,-6.7;
move -21,-485.7,7.5,-13.2,11.1,-6.6;
move -24,-485,7.5,-13.2,11.2,-6.5;
move -26,-484.2,7.6,-13.6,11.3,-6.5;
move -28,-483.4,7.7,-14,11.4,-6.4;
move -30,-482.5,7.7,-14.4,11.5,-6.4;
move -33,-481.6,7.7,-14.8,11.5,-6.3;
move -35,-480.6,7.8,-15.2,11.6,-6.2;
move -37,-479.5,7.8,-15.2,11.7,-6.2;
move -39,-478.4,7.9,-15.6,11.8,-6.1;
move -42,-477.2,7.9,-16,11.8,-6;
move -44,-475.9,8,-16.4,11.9,-6;
move -46,-474.5,8,-16.4,12,-5.9;
move -48,-473.1,8.1,-16.8,12.1,-5.8;
move -51,-471.5,8.1,-17.2,12.1,-5.8;
move -53,-469.9,8.1,-17.6,12.2,-5.7;
move -55,-468.2,8.2,-17.6,12.3,-5.6;
move -57,-466.4,8.2,-18,12.4,-5.6;
move -60,-464.5,8.3,-18.4,12.4,-5.5;
move -62,-462.6,8.3,-18.8,12.5,-5.4;
move -64,-460.6,8.4,-19.2,12.6,-5.4;
move -66,-458.5,8.4,-19.2,12.6,-5.3;
move -68,-456.3,8.5,-19.6,12.7,-5.2;
move -70,-454.1,8.5,-19.6,12.8,-5.1;
move -72,-451.8,8.5,-20,12.8,-5.1;
move -74,-449.5,8.5,-20.4,12.9,-5;
move -75,-447.2,8.6,-20.4,13,-4.9;
move -77,-444.8,8.6,-20.8,13,-4.9;
move -79,-442.4,8.6,-21.2,13.1,-4.8;
move -81,-439.9,8.7,-21.2,13.1,-4.7;
move -83,-437.4,8.7,-21.6,13.2,-4.6;
move -85,-435,8.7,-21.6,13.3,-4.6;
move -87,-432.5,8.7,-22,13.3,-4.5;
move -89,-430,8.8,-22.4,13.4,-4.4;
move -90,-427.5,8.8,-22.8,13.4,-4.4;
move -92,-425,8.8,-22.8,13.5,-4.3;
move -93,-422.5,8.8,-23.2,13.5,-4.2;
move -95,-420.1,8.8,-23.2,13.6,-4.1;
move -96,-417.6,8.9,-23.6,13.7,-4.1;
move -98,-415.2,8.9,-23.6,13.7,-4;
move -99,-412.8,8.9,-23.6,13.8,-3.9;
move -100,-410.4,8.9,-24,13.8,-3.8;
move -101,-408,8.9,-24,13.9,-3.8;
move -101,-405.7,8.9,-24,13.9,-3.7;
move -102,-403.4,9,-24.4,13.9,-3.6;
move -103,-401.1,9,-24.4,14,-3.5;
move -104,-398.8,9,-24.4,14,-3.4;
move -104,-396.5,9,-24.4,14.1,-3.4;
move -105,-394.3,9.1,-24.4,14.1,-3.3;
move -105,-392,9.1,-24.4,14.2,-3.2;
move -105,-389.7,9.1,-24.8,14.2,-3.1;
move -105,-387.4,9.2,-24.8,14.2,-3.1;
move -105,-385.1,9.2,-24.8,14.3,-3;
move -105,-382.8,9.2,-24.8,14.3,-2.9;
move -105,-380.5,9.2,-24.8,14.4,-2.8;
move -105,-378.1,9.3,-24.4,14.4,-2.7;
move -105,-375.8,9.3,-24.4,14.4,-2.7;
move -104,-373.4,9.3,-24.4,14.5,-2.6;
move -104,-371,9.3,-24.4,14.5,-2.5;
move -103,-368.6,9.4,-24.4,14.5,-2.4;
move -103,-366.2,9.4,-24.4,14.6,-2.3;
move -102,-363.8,9.4,-24.4,14.6,-2.3;
move -101,-361.4,9.4,-24,14.6,-2.2;
move -100,-359,9.4,-24,14.6,-2.1;
move -100,-356.6,9.4,-23.6,14.7,-2;
move -99,-354.3,9.4,-23.6,14.7,-1.9;
move -98,-351.9,9.4,-23.6,14.7,-1.9;
move -97,-349.6,9.4,-23.6,14.7,-1.8;
move -96,-347.3,9.4,-23.2,14.8,-1.7;
move -94,-345.1,9.4,-23.2,14.8,-1.6;
move -93,-342.9,9.4,-22.8,14.8,-1.5;
move -92,-340.7,9.4,-22.8,14.8,-1.5;
move -91,-338.6,9.4,-22.8,14.8,-1.4;
move -90,-336.6,9.4,-22.4,14.9,-1.3;
move -88,-334.6,9.4,-22.4,14.9,-1.2;
move -87,-332.6,9.4,-22,14.9,-1.1;
move -86,-330.7,9.4,-22,14.9,-1;
move -84,-328.9,9.4,-21.6,14.9,-1;
move -83,-327.1,9.4,-21.6,14.9,-0.9;
move -81,-325.4,9.3,-21.2,14.9,-0.8;
move -80,-323.7,9.3,-21.2,15,-0.7;
move -78,-322,9.3,-20.8,15,-0.6;
move -77,-320.4,9.3,-20.8,15,-0.5;
move -75,-318.9,9.2,-20.4,15,-0.5;
move -73,-317.3,9.2,-20.4,15,-0.4;
move -71,-315.8,9.1,-20,15,-0.3;
move -69,-314.2,9.1,-19.6,15,-0.2;
move -68,-312.7,9.1,-19.6,15,-0.1;
move -66,-311.2,9,-19.2,15,-0;
move -64,-309.7,9,-18.8,15,0;
move -62,-308.1,8.9,-18.8,15,0.1;
move -59,-306.6,8.9,-18.4,15,0.2;
move -57,-305,8.8,-18,15,0.3;
move -55,-303.4,8.7,-17.6,15,0.4;
move -53,-301.9,8.7,-17.6,15,0.4;
move -51,-300.2,8.6,-17.2,15,0.5;
move -49,-298.6,8.5,-16.8,15,0.6;
move -46,-296.9,8.5,-16.4,15,0.7;
move -44,-295.3,8.4,-16.4,15,0.8;
move -42,-293.6,8.3,-16,15,0.9;
move -39,-291.9,8.2,-15.6,14.9,0.9;
move -37,-290.1,8.1,-15.2,14.9,1;
move -35,-288.4,8,-14.8,14.9,1.1;
move -32,-286.6,7.9,-14.8,14.9,1.2;
move -30,-284.9,7.8,-14.4,14.9,1.3;
move -28,-283.2,7.7,-14,14.9,1.3;
move -25,-281.5,7.6,-13.6,14.9,1.4;
move -23,-279.9,7.4,-13.2,14.8,1.5;
move -20,-278.2,7.3,-13.2,14.8,1.6;
move -18,-276.6,7.2,-12.8,14.8,1.7;
move -15,-275.1,7.1,-12.4,14.8,1.8;
move -13,-273.6,6.9,-12,14.8,1.8;
move -11,-272.1,6.8,-11.6,14.7,1.9;
move -8,-270.7,6.7,-11.2,14.7,2;
move -6,-269.5,6.5,-10.8,14.7,2.1;
move -3,-268.2,6.3,-10.8,14.7,2.2;
move -1,-267.1,6.2,-10.4,14.6,2.2;
move 2,-266,6,-10,14.6,2.3;
move 4,-265.1,5.8,-9.6,14.6,2.4;
move 6,-264.3,5.7,-9.2,14.5,2.5;
move 8,-263.5,5.5,-9.2,14.5,2.6;
move 11,-262.9,5.3,-8.8,14.5,2.6;
move 13,-262.4,5.2,-8.4,14.4,2.7;
move 15,-262.1,5,-8,14.4,2.8;
move 17,-261.8,4.8,-8,14.4,2.9;
move 19,-261.6,4.6,-7.6,14.3,3;
move 22,-261.6,4.4,-7.2,14.3,3;
move 24,-261.7,4.3,-7.2,14.3,3.1;
move 26,-261.9,4.1,-6.8,14.2,3.2;
move 28,-262.2,3.9,-6.4,14.2,3.3;
move 30,-262.5,3.7,-6,14.1,3.3;
move 32,-263,3.5,-5.6,14.1,3.4;
move 35,-263.5,3.3,-5.6,14.1,3.5;
move 37,-264,3.1,-5.2,14,3.6;
move 39,-264.6,3,-4.8,14,3.7;
move 41,-265.2,2.8,-4.8,13.9,3.7;
move 43,-265.7,2.6,-4.4,13.9,3.8;
move 44,-266.3,2.4,-4,13.8,3.9;
move 46,-266.8,2.3,-4,13.8,4;
move 48,-267.2,2.1,-3.6,13.7,4;
move 50,-267.6,1.9,-3.6,13.7,4.1;
move 52,-267.9,1.7,-3.2,13.6,4.2;
move 53,-268.1,1.5,-2.8,13.6,4.3;
move 55,-268.2,1.4,-2.8,13.5,4.3;
move 57,-268.3,1.2,-2.4,13.5,4.4;
move 58,-268.2,1,-2.4,13.4,4.5;
move 60,-268,0.8,-2,13.4,4.6;
move 61,-267.8,0.6,-1.6,13.3,4.6;
move 63,-267.5,0.4,-1.6,13.2,4.7;
move 64,-267.1,0.3,-1.6,13.2,4.8;
move 65,-266.6,0.1,-1.2,13.1,4.9;
move 67,-266.1,-0,-1.2,13.1,4.9;
move 68,-265.6,-0.2,-1.2,13,5;
move 69,-265,-0.3,-0.8,12.9,5.1;
move 70,-264.4,-0.5,-0.8,12.9,5.1;
move 71,-263.7,-0.6,-0.4,12.8,5.2;
move 73,-263.1,-0.8,-0.4,12.7,5.3;
move 74,-262.5,-0.9,-0,12.7,5.4;
move 75,-262,-1.1,0,12.6,5.4;
move 76,-261.4,-1.2,0,12.5,5.5;
move 77,-261,-1.3,0.4,12.5,5.6;
move 78,-260.5,-1.4,0.4,12.4,5.6;
move 79,-260.2,-1.5,0.4,12.3,5.7;
move 80,-259.9,-1.6,0.8,12.3,5.8;
move 81,-259.7,-1.7,0.8,12.2,5.8;
move 82,-259.6,-1.8,0.8,12.1,5.9;
move 83,-259.5,-1.9,0.8,12,6;
move 84,-259.6,-2,1.2,12,6;
move 85,-259.8,-2.1,1.2,11.9,6.1;
move 86,-260,-2.2,1.6,11.8,6.2;
move 87,-260.3,-2.3,1.6,11.7,6.2;
move 88,-260.6,-2.4,1.6,11.6,6.3;
move 89,-261.1,-2.5,1.6,11.6,6.3;
move 90,-261.6,-2.5,2,11.5,6.4;
move 91,-262.1,-2.6,2,11.4,6.5;
move 92,-262.7,-2.7,2.4,11.3,6.5;
move 93,-263.3,-2.8,2.4,11.2,6.6;
move 93,-264,-2.8,2.8,11.2,6.7;
move 94,-264.6,-2.9,2.8,11.1,6.7;
move 95,-265.3,-2.9,2.8,11,6.8;
move 95,-266.1,-3,2.8,10.9,6.8;
move 96,-266.8,-3.1,2.8,10.8,6.9;
move 96,-267.6,-3.1,2.8,10.7,7;
move 96,-268.3,-3.2,2.8,10.6,7;
move 96,-269.1,-3.3,2.8,10.6,7.1;
move 97,-269.8,-3.3,2.8,10.5,7.1;
move 97,-270.5,-3.4,2.8,10.4,7.2;
move 97,-271.2,-3.4,3.2,10.3,7.2;
move 98,-271.8,-3.5,3.2,10.2,7.3;
move 98,-272.5,-3.5,2.8,10.1,7.4;
move 98,-273,-3.5,3.2,10,7.4;
move 98,-273.5,-3.6,3.2,9.9,7.5;
move 98,-274,-3.6,3.2,9.8,7.5;
move 99,-274.5,-3.7,3.2,9.7,7.6;
move 99,-274.9,-3.7,3.2,9.6,7.6;
move 99,-275.3,-3.7,3.2,9.5,7.7;
move 99,-275.6,-3.8,3.2,9.4,7.7;
move 99,-275.9,-3.8,3.2,9.3,7.8;
move 99,-276.2,-3.9,3.2,9.2,7.8;
move 99,-276.5,-3.9,3.2,9.1,7.9;
move 99,-276.7,-4,3.2,9,7.9;
move 99,-276.9,-4,3.2,8.9,8;
move 99,-277.1,-4,3.2,8.8,8;
move 99,-277.3,-4.1,3.2,8.7,8.1;
move 98,-277.4,-4.1,3.2,8.6,8.1;
move 98,-277.6,-4.1,3.2,8.5,8.2;
move 98,-277.7,-4.2,3.2,8.4,8.2;
move 98,-277.9,-4.2,3.2,8.3,8.3;
move 97,-278,-4.3,2.8,8.2,8.3;
move 97,-278.1,-4.3,2.8,8.1,8.4;
move 97,-278.1,-4.3,2.8,8,8.4;
move 96,-278.1,-4.3,2.8,7.9,8.4;
move 96,-278.1,-4.3,2.8,7.8,8.5;
move 96,-278,-4.3,2.8,7.7,8.5;
move 95,-277.9,-4.4,2.8,7.6,8.6;
move 95,-277.8,-4.4,2.8,7.5,8.6;
move 95,-277.6,-4.4,2.8,7.4,8.7;
move 94,-277.4,-4.4,2.4,7.3,8.7;
move 94,-277.1,-4.4,2.4,7.2,8.7;
move 93,-276.9,-4.4,2.4,7,8.8;
move 93,-276.7,-4.4,2.4,6.9,8.8;
move 93,-276.4,-4.4,2.4,6.8,8.8;
move 92,-276.2,-4.4,2.4,6.7,8.9;
move 92,-275.9,-4.4,2.4,6.6,8.9;
move 91,-275.7,-4.4,2,6.5,9;
move 91,-275.6,-4.4,2,6.4,9;
move 90,-275.5,-4.4,2,6.3,9;
move 90,-275.6,-4.3,2,6.1,9.1;
move 89,-275.9,-4.3,2,6,9.1;
move 89,-276.2,-4.3,2,5.9,9.1;
move 88,-276.5,-4.3,1.6,5.8,9.2;
move 88,-276.9,-4.3,1.6,5.7,9.2;
move 87,-277.4,-4.2,1.6,5.6,9.2;
move 87,-277.9,-4.2,1.6,5.5,9.3;
move 86,-278.5,-4.1,1.6,5.3,9.3;
move 86,-279.2,-4.1,1.2,5.2,9.3;
move 85,-280,-4,1.2,5.1,9.4;
move 84,-280.8,-4,1.2,5,9.4;
move 84,-281.7,-3.9,1.2,4.9,9.4;
move 83,-282.6,-3.8,1.2,4.8,9.5;
move 83,-283.5,-3.8,1.2,4.6,9.5;
move 82,-284.4,-3.7,0.8,4.5,9.5;
move 81,-285.2,-3.6,0.8,4.4,9.5;
move 81,-285.9,-3.5,0.8,4.3,9.6;
move 80,-286.5,-3.4,0.8,4.2,9.6;
move 79,-286.9,-3.3,0.4,4,9.6;
move 79,-287.2,-3.2,0.4,3.9,9.7;
move 78,-287.2,-3.1,0.4,3.8,9.7;
move 78,-287.1,-3,0.4,3.7,9.7;
move 77,-286.7,-2.9,0,3.6,9.7;
move 77,-286.1,-2.8,0,3.4,9.7;
move 76,-285.2,-2.6,0,3.3,9.8;
move 76,-284.1,-2.4,0,3.2,9.8;
move 76,-282.8,-2.3,0,3.1,9.8;
move 76,-281.3,-2.1,0,2.9,9.8;
move 75,-279.6,-2,-0,2.8,9.8;
move 75,-277.7,-1.8,-0,2.7,9.9;
move 75,-275.7,-1.7,-0,2.6,9.9;
move 75,-273.6,-1.5,-0,2.4,9.9;
move 75,-271.4,-1.3,-0,2.3,9.9;
move 75,-269.3,-1.2,-0,2.2,9.9;
move 75,-267.1,-1,-0,2.1,9.9;
move 75,-265,-0.8,-0,2,9.9;
move 76,-263,-0.6,-0,1.8,9.9;
move 76,-261,-0.4,-0,1.7,9.9;
move 76,-259.2,-0.2,-0,1.6,9.9;
move 76,-257.5,-0,0,1.5,10;
move 77,-255.9,0.2,0,1.3,10;
move 77,-254.5,0.4,0,1.2,10;
move 77,-253.2,0.6,0.4,1.1,10;
move 78,-252.1,0.8,0.4,1,10;
move 79,-251,1,0.4,0.8,10;
move 79,-250.1,1.2,0.4,0.7,10;
move 80,-249.3,1.4,0.4,0.6,10;
move 81,-248.5,1.6,0.8,0.5,10;
move 82,-247.8,1.8,0.8,0.3,10;
move 83,-247.2,2.1,0.8,0.2,10;
move 84,-246.5,2.2,1.2,0.1,10;
move 85,-245.9,2.4,1.2,-0,10;
move 86,-245.3,2.7,1.6,-0.2,10;
move 87,-244.9,2.9,1.6,-0.3,10;
move 88,-244.5,3.1,1.6,-0.4,10;
move 90,-244.1,3.3,2,-0.5,10;
move 91,-243.6,3.5,2,-0.7,10;
move 92,-243.2,3.6,2.4,-0.8,10;
move 94,-242.8,3.8,2.4,-0.9,10;
move 95,-242.4,4,2.8,-1,10;
move 97,-241.9,4.2,2.8,-1.2,10;
move 98,-241.5,4.3,3.2,-1.3,10;
move 99,-241.2,4.5,3.2,-1.4,10;
move 101,-240.9,4.7,3.6,-1.5,10;
move 102,-240.6,4.9,3.6,-1.7,9.9;
move 104,-240.5,5,3.6,-1.8,9.9;
move 105,-240.4,5.2,4,-1.9,9.9;
move 107,-240.3,5.4,4.4,-2,9.9;
move 108,-240.4,5.5,4.4,-2.2,9.9;
move 110,-240.6,5.6,4.8,-2.3,9.9;
move 112,-240.8,5.8,4.8,-2.4,9.9;
move 113,-241.2,5.9,5.2,-2.5,9.9;
move 115,-241.6,6,5.6,-2.7,9.9;
move 116,-242.2,6.1,5.6,-2.8,9.8;
move 118,-242.9,6.2,6,-2.9,9.8;
move 119,-243.6,6.3,6,-3,9.8;
move 121,-244.5,6.4,6.4,-3.1,9.8;
move 122,-245.5,6.4,6.4,-3.3,9.8;
move 123,-246.6,6.5,6.4,-3.4,9.7;
move 124,-247.7,6.6,6.8,-3.5,9.7;
move 125,-248.9,6.7,6.8,-3.6,9.7;
move 126,-250.2,6.7,6.8,-3.8,9.7;
move 127,-251.5,6.7,7.2,-3.9,9.7;
move 128,-252.9,6.7,7.2,-4,9.6;
move 129,-254.3,6.7,7.2,-4.1,9.6;
move 130,-255.8,6.7,7.6,-4.2,9.6;
move 131,-257.3,6.7,7.6,-4.4,9.5;
move 131,-258.9,6.7,7.6,-4.5,9.5;
move 132,-260.6,6.7,7.6,-4.6,9.5;
move 133,-262.2,6.7,8,-4.7,9.5;
move 133,-263.9,6.7,8,-4.8,9.4;
move 134,-265.7,6.6,8,-4.9,9.4;
move 134,-267.5,6.6,8,-5.1,9.4;
move 134,-269.3,6.5,8,-5.2,9.3;
move 134,-271.2,6.5,8,-5.3,9.3;
move 134,-273.1,6.5,8.4,-5.4,9.3;
move 134,-275,6.4,8.4,-5.5,9.2;
move 134,-277,6.3,8,-5.7,9.2;
move 133,-278.9,6.3,8,-5.8,9.2;
move 133,-280.9,6.2,8,-5.9,9.1;
move 132,-282.9,6.1,7.6,-6,9.1;
move 132,-284.9,6.1,7.6,-6.1,9;
move 131,-286.9,6,7.6,-6.2,9;
move 130,-288.9,5.9,7.6,-6.3,9;
move 129,-290.8,5.9,7.6,-6.5,8.9;
move 128,-292.8,5.8,7.2,-6.6,8.9;
move 127,-294.7,5.7,7.2,-6.7,8.9;
move 125,-296.5,5.6,6.8,-6.8,8.8;
move 124,-298.3,5.5,6.8,-6.9,8.8;
move 122,-299.9,5.4,6.4,-7,8.7;
move 121,-301.5,5.3,6,-7.1,8.7;
move 119,-303,5.2,6,-7.2,8.7;
move 117,-304.5,5.1,5.6,-7.3,8.6;
move 115,-305.8,5.1,5.6,-7.4,8.6;
move 113,-307,5,5.2,-7.6,8.5;
move 111,-308.1,4.9,4.8,-7.7,8.5;
move 110,-309.1,4.8,4.8,-7.8,8.5;
move 108,-310,4.7,4.4,-7.9,8.4;
move 106,-310.8,4.6,4,-8,8.4;
move 103,-311.6,4.6,4,-8.1,8.3;
move 101,-312.2,4.5,3.6,-8.2,8.3;
move 99,-312.7,4.4,3.2,-8.3,8.2;
move 97,-313.1,4.4,2.8,-8.4,8.2;
move 95,-313.4,4.3,2.8,-8.5,8.1;
move 93,-313.5,4.3,2.4,-8.6,8.1;
move 91,-313.5,4.2,2,-8.7,8;
move 88,-313.4,4.1,1.6,-8.8,8;
move 86,-313.1,4.1,1.6,-8.9,7.9;
move 84,-312.8,4.1,1.2,-9,7.9;
move 82,-312.3,4,0.8,-9.1,7.8;
move 80,-311.7,4,0.4,-9.2,7.8;
move 78,-311,4,0.4,-9.3,7.7;
move 76,-310.1,4,0,-9.4,7.7;
move 73,-309.1,4,-0.4,-9.5,7.6;
move 71,-308.1,4,-0.4,-9.6,7.6;
move 70,-306.9,4,-0.8,-9.7,7.5;
move 68,-305.7,4,-1.2,-9.8,7.5;
move 66,-304.4,4,-1.6,-9.9,7.4;
move 64,-303.1,4,-1.6,-10,7.4;
move 62,-301.8,4,-2,-10.1,7.3;
move 61,-300.4,4,-2,-10.2,7.3;
move 59,-299.1,4.1,-2,-10.3,7.2;
move 57,-297.7,4.1,-2.4,-10.3,7.1;
move 56,-296.4,4.2,-2.8,-10.4,7.1;
move 54,-295.1,4.2,-3.2,-10.5,7;
move 53,-293.9,4.3,-3.2,-10.6,7;
move 51,-292.8,4.3,-3.2,-10.7,6.9;
move 50,-291.8,4.4,-3.6,-10.8,6.8;
move 49,-290.9,4.5,-3.6,-10.9,6.8;
move 48,-290,4.6,-3.6,-11,6.7;
move 47,-289.3,4.6,-4,-11,6.7;
move 46,-288.7,4.7,-4.4,-11.1,6.6;
move 45,-288.2,4.8,-4.4,-11.2,6.5;
move 44,-287.8,4.9,-4.4,-11.3,6.5;
move 43,-287.6,5,-4.4,-11.4,6.4;
move 43,-287.4,5.1,-4.4,-11.5,6.4;
move 42,-287.4,5.3,-4.4,-11.5,6.3;
move 42,-287.5,5.4,-4.4,-11.6,6.2;
move 42,-287.6,5.5,-4.8,-11.7,6.2;
move 41,-287.9,5.6,-4.8,-11.8,6.1;
move 41,-288.1,5.8,-4.8,-11.9,6;
move 41,-288.4,5.9,-4.8,-11.9,6;
move 41,-288.7,6,-4.8,-12,5.9;
move 41,-288.9,6.1,-4.8,-12.1,5.8;
move 41,-289,6.2,-4.8,-12.2,5.8;
move 41,-289.1,6.4,-4.8,-12.2,5.7;
move 42,-289,6.5,-4.8,-12.3,5.6;
move 42,-288.8,6.6,-4.8,-12.4,5.6;
move 43,-288.3,6.7,-4.4,-12.4,5.5;
move 44,-287.6,6.8,-4.4,-12.5,5.4;
move 45,-286.7,7,-4,-12.6,5.4;
move 46,-285.5,7.1,-4,-12.6,5.3;
move 47,-284.1,7.2,-4,-12.7,5.2;
move 48,-282.5,7.4,-4,-12.8,5.1;
move 49,-280.6,7.5,-3.6,-12.8,5.1;
move 50,-278.6,7.6,-3.6,-12.9,5;
move 52,-276.3,7.7,-3.2,-13,4.9;
move 53,-273.9,7.8,-3.2,-13,4.9;
move 55,-271.4,7.9,-2.8,-13.1,4.8;
move 56,-268.8,8.1,-2.8,-13.2,4.7;
move 58,-266.1,8.2,-2.4,-13.2,4.6;
move 60,-263.4,8.3,-2,-13.3,4.6;
move 62,-260.8,8.4,-2,-13.3,4.5;
move 64,-258.2,8.5,-1.6,-13.4,4.4;
move 66,-255.8,8.6,-1.2,-13.4,4.4;
move 68,-253.5,8.7,-1.2,-13.5,4.3;
move 70,-251.5,8.8,-0.8,-13.6,4.2;
move 73,-249.6,8.9,-0.4,-13.6,4.1;
move 75,-248,9,-0,-13.7,4.1;
move 77,-246.6,9.1,0.4,-13.7,4;
move 80,-245.5,9.1,0.4,-13.8,3.9;
move 82,-244.6,9.2,0.8,-13.8,3.8;
move 85,-244,9.2,1.2,-13.9,3.8;
move 87,-243.7,9.3,1.6,-13.9,3.7;
move 90,-243.6,9.4,2,-14,3.6;
move 93,-243.7,9.4,2.4,-14,3.5;
move 95,-244,9.5,2.8,-14,3.4;
move 98,-244.5,9.5,3.2,-14.1,3.4;
move 101,-245.2,9.5,3.6,-14.1,3.3;
move 103,-246.1,9.5,4,-14.2,3.2;
move 106,-247.1,9.6,4,-14.2,3.1;
move 109,-248.1,9.6,4.4,-14.2,3.1;
move 111,-249.3,9.6,4.8,-14.3,3;
move 114,-250.6,9.6,5.2,-14.3,2.9;
move 117,-252,9.6,5.6,-14.4,2.8;
move 120,-253.5,9.6,6,-14.4,2.7;
move 122,-255.2,9.6,6.4,-14.4,2.7;
move 125,-256.9,9.6,6.8,-14.5,2.6;
move 128,-258.7,9.6,7.2,-14.5,2.5;
move 131,-260.5,9.5,7.6,-14.5,2.4;
move 134,-262.4,9.5,8,-14.6,2.3;
move 137,-264.3,9.5,8.4,-14.6,2.3;
move 140,-266.3,9.4,8.8,-14.6,2.2;
move 143,-268.3,9.4,9.2,-14.6,2.1;
move 145,-270.4,9.3,9.6,-14.7,2;
move 148,-272.6,9.3,10,-14.7,1.9;
move 151,-274.8,9.2,10.4,-14.7,1.9;
move 153,-277,9.2,10.8,-14.7,1.8;
move 156,-279.2,9.1,10.8,-14.8,1.7;
move 158,-281.5,9.1,11.2,-14.8,1.6;
move 161,-283.7,9,11.6,-14.8,1.5;
move 163,-286,9,12,-14.8,1.5;
move 166,-288.3,8.9,12.4,-14.8,1.4;
move 168,-290.6,8.8,12.8,-14.9,1.3;
move 171,-292.8,8.8,13.2,-14.9,1.2;
move 173,-295,8.7,13.2,-14.9,1.1;
move 175,-297.1,8.7,13.6,-14.9,1;
move 177,-299.2,8.6,14,-14.9,1;
move 179,-301.2,8.6,14,-14.9,0.9;
move 181,-303.2,8.5,14.4,-14.9,0.8;
move 183,-305.1,8.4,14.8,-15,0.7;
move 185,-306.9,8.4,15.2,0,0.6;
move 187,-308.6,8.3,15.2,0,0.5;
move 189,-310.3,8.3,15.6,0,0.5;
move 191,-312,8.3,16,0,0.4;
move 192,-313.5,8.2,16,0,0.3;
move 194,-315.1,8.2,16.4,0,0.2;
move 195,-316.6,8.1,16.4,0,0.1;
move 197,-318.2,8.1,16.4,0,0;
move 198,-319.8,8,16.8,0,-0;
move 199,-321.3,8,16.8,0,-0.1;
move 200,-323,8,17.2,0,-0.2;
move 201,-324.6,7.9,17.2,0,-0.3;
move 202,-326.3,7.9,17.2,0,-0.4;
move 203,-328.1,7.9,17.2,0,-0.5;
move 204,-330,7.8,17.6,0,-0.5;
move 205,-332,7.8,17.6,0,-0.6;
move 206,-334,7.8,17.6,0,-0.7;
move 207,-336,7.8,18,0,-0.8;
move 208,-338.1,7.8,18,0,-0.9;
move 209,-340.3,7.8,18.4,0,-1;
move 209,-342.6,7.8,18.4,0,-1;
move 210,-344.9,7.8,18.4,0,-1.1;
move 211,-347.3,7.7,18.4,0,-1.2;
move 211,-349.6,7.8,18.4,0,-1.3;
move 212,-352,7.8,18.8,0,-1.4;
move 212,-354.3,7.8,18.8,0,-1.4;
move 212,-356.6,7.8,18.8,0,-1.5;
move 212,-359,7.8,18.8,0,-1.6;
move 212,-361.3,7.8,18.8,0,-1.7;
move 212,-363.7,7.9,18.8,0,-1.8;
move 211,-366,7.9,18.4,0,-1.9;
move 211,-368.2,7.9,18.4,0,-1.9;
move 210,-370.4,7.9,18.4,0,-2;
move 209,-372.5,7.9,18.4,0,-2.1;
move 208,-374.6,7.9,18,0,-2.2;
move 207,-376.6,8,18,0,-2.3;
move 206,-378.6,8,18,0,-2.3;
move 205,-380.6,8,17.6,0,-2.4;
move 203,-382.4,8,17.6,0,-2.5;
move 202,-384.2,8,17.6,0,-2.6;
move 200,-386,8.1,17.2,0,-2.7;
move 199,-387.7,8.1,16.8,0,-2.7;
move 197,-389.3,8.1,16.4,0,-2.8;
move 196,-391,8.2,16,0,-2.9;
move 194,-392.6,8.2,16,0,-3;
move 192,-394.2,8.2,16,0,-3.1;
move 191,-395.7,8.3,15.6,0,-3.1;
move 189,-397.2,8.3,15.6,0,-3.2;
move 187,-398.7,8.3,15.2,0,-3.3;
move 186,-400.2,8.3,15.2,0,-3.4;
move 184,-401.7,8.3,14.8,-14.1,-3.4;
move 182,-403.3,8.3,14.4,-14.1,-3.5;
move 181,-404.8,8.3,14.4,-14,-3.6;
move 179,-406.3,8.3,14,-14,-3.7;
move 177,-407.9,8.3,14,-13.9,-3.7;
move 175,-409.6,8.3,13.6,-13.9,-3.8;
move 173,-411.2,8.3,13.2,-13.8,-3.9;
move 172,-412.9,8.3,13.2,-13.8,-4;
move 170,-414.6,8.2,12.8,-13.7,-4;
move 168,-416.3,8.2,12.4,-13.7,-4.1;
move 166,-418,8.1,12.4,-13.6,-4.2;
move 164,-419.7,8.1,12,-13.6,-4.3;
move 163,-421.5,8,12,-13.5,-4.3;
move 161,-423.2,8,11.6,-13.5,-4.4;
move 159,-425,7.9,11.6,-13.4,-4.5;
move 157,-426.7,7.8,11.2,-13.3,-4.6;
move 155,-428.5,7.7,10.8,-13.3,-4.6;
move 153,-430.1,7.6,10.4,-13.2,-4.7;
move 150,-431.8,7.5,10.4,-13.2,-4.8;
move 148,-433.4,7.4,10,-13.1,-4.9;
move 146,-434.9,7.3,9.6,-13,-4.9;
move 144,-436.3,7.2,9.2,-13,-5;
move 141,-437.7,7.1,8.8,-12.9,-5.1;
move 139,-438.9,6.9,8.4,-12.9,-5.1;
move 137,-439.9,6.8,8.4,-12.8,-5.2;
move 135,-440.9,6.6,8,-12.7,-5.3;
move 134,-441.7,6.5,7.6,-12.7,-5.4;
move 132,-442.3,6.3,7.6,-12.6,-5.4;
move 131,-442.8,6.2,7.6,-12.5,-5.5;
move 129,-443.1,6,7.2,-12.5,-5.6;
move 128,-443.2,5.8,7.2,-12.4,-5.6;
move 126,-443.3,5.6,6.8,-12.3,-5.7;
move 125,-443.1,5.4,6.8,-12.2,-5.8;
move 124,-442.8,5.2,6.4,-12.2,-5.8;
move 122,-442.3,5,6.4,-12.1,-5.9;
move 121,-441.7,4.9,6.4,-12,-6;
move 120,-441,4.7,6,-11.9,-6;
move 119,-440.1,4.5,6,-11.9,-6.1;
move 117,-439.2,4.3,5.6,-11.8,-6.2;
move 116,-438.1,4,5.6,-11.7,-6.2;
move 115,-437,3.8,5.2,-11.6,-6.3;
move 114,-435.8,3.6,5.2,-11.6,-6.3;
move 113,-434.5,3.3,5.2,-11.5,-6.4;
move 111,-433,3.1,4.8,-11.4,-6.5;
move 110,-431.4,2.9,4.8,-11.3,-6.5;
move 109,-429.7,2.6,4.4,-11.2,-6.6;
move 108,-428.1,2.4,4.4,-11.1,-6.7;
move 107,-426.5,2.1,4.4,-11.1,-6.7;
move 106,-424.9,1.9,4,-11,-6.8;
move 106,-423.2,1.7,4,-10.9,-6.8;
move 105,-421.5,1.4,4,-10.8,-6.9;
move 104,-419.9,1.2,4,-10.7,-7;
move 104,-418.3,1,3.6,-10.6,-7;
move 103,-416.7,0.7,3.6,-10.5,-7.1;
move 103,-415.2,0.5,3.6,-10.5,-7.1;
move 102,-413.8,0.2,3.6,-10.4,-7.2;
move 102,-412.5,0,3.6,-10.3,-7.2;
move 101,-411.4,-0.2,3.6,-10.2,-7.3;
move 101,-410.4,-0.4,3.6,-10.1,-7.4;
move 100,-409.5,-0.6,3.6,-10,-7.4;
move 99,-408.9,-0.8,3.2,-9.9,-7.5;
move 99,-408.6,-1,3.2,-9.8,-7.5;
move 98,-408.5,-1.2,3.2,-9.7,-7.6;
move 97,-408.7,-1.4,3.2,-9.6,-7.6;
move 96,-409.3,-1.6,2.8,-9.5,-7.7;
move 94,-410.3,-1.8,2.8,-9.4,-7.7;
move 93,-411.6,-1.9,2.4,-9.3,-7.8;
move 92,-413.4,-2.1,2.4,-9.2,-7.8;
move 90,-415.6,-2.2,2,-9.1,-7.9;
move 89,-418.1,-2.4,2,-9,-7.9;
move 87,-421,-2.5,1.6,-8.9,-8;
move 85,-424.3,-2.6,1.2,-8.8,-8;
move 83,-427.9,-2.7,1.2,-8.7,-8.1;
move 81,-431.9,-2.8,0.8,-8.6,-8.1;
move 79,-436.1,-3,0.8,-8.5,-8.2;
move 77,-440.6,-3.1,0.4,-8.4,-8.2;
move 75,-445.3,-3.2,-0,-8.3,-8.3;
move 72,-450.1,-3.2,-0.4,-8.2,-8.3;
move 70,-455,-3.3,-0.8,-8.1,-8.4;
move 67,-459.8,-3.3,-0.8,-8,-8.4;
move 64,-464.6,-3.4,-1.2,-7.9,-8.4;
move 61,-469.2,-3.4,-1.6,-7.8,-8.5;
move 58,-473.6,-3.4,-2.4,-7.7,-8.5;
move 55,-477.8,-3.4,-2.8,-7.6,-8.6;
move 51,-481.5,-3.4,-3.2,-7.5,-8.6;
move 48,-484.9,-3.4,-3.6,-7.4,-8.7;
move 44,-487.8,-3.4,-4,-7.3,-8.7;
move 40,-490.2,-3.3,-4.8,-7.1,-8.7;
move 36,-492.1,-3.3,-5.2,-7,-8.8;
move 32,-493.3,-3.2,-6,-6.9,-8.8;
move 28,-494.1,-3.2,-6.4,-6.8,-8.9;
move 24,-494.2,-3.1,-7.2,-6.7,-8.9;
move 20,-493.7,-3,-7.6,-6.6,-8.9;
move 16,-492.8,-2.9,-8,-6.5,-9;
move 12,-491.3,-2.8,-8.8,-6.4,-9;
move 8,-489.2,-2.7,-9.2,-6.2,-9;
move 4,-486.5,-2.6,-9.6,-6.1,-9.1;
move 0,-483.3,-2.5,-10.4,-6,-9.1;
move -4,-479.7,-2.4,-10.8,-5.9,-9.2;
move -8,-475.6,-2.2,-11.6,-5.8,-9.2;
move -12,-471.1,-2.1,-12,-5.7,-9.2;
move -16,-466.3,-2,-12.4,-5.6,-9.3;
move -19,-461.1,-1.9,-13.2,-5.4,-9.3;
move -22,-455.5,-1.7,-13.6,-5.3,-9.3;
move -25,-449.7,-1.6,-14,-5.2,-9.4;
move -28,-443.6,-1.4,-14.4,-5.1,-9.4;
move -31,-437.2,-1.3,-14.8,-5,-9.4;
move -33,-430.6,-1.1,-14.8,-4.9,-9.4;
move -36,-423.7,-1,-15.2,-4.7,-9.5;
move -38,-416.7,-0.8,-15.6,-4.6,-9.5;
move -40,-409.5,-0.7,-15.6,-4.5,-9.5;
move -42,-402.2,-0.5,-16,-4.4,-9.6;
move -43,-394.7,-0.4,-16.4,-4.3,-9.6;
move -45,-387.3,-0.2,-16.4,-4.1,-9.6;
move -47,-379.9,-0,-16.8,-4,-9.6;
move -48,-372.4,0.1,-16.8,-3.9,-9.7;
move -49,-365.1,0.3,-17.2,-3.8,-9.7;
move -50,-358,0.4,-17.2,-3.7,-9.7;
move -51,-351,0.6,-17.6,-3.5,-9.7;
move -52,-344.4,0.8,-17.6,-3.4,-9.8;
move -52,-338,0.9,-17.6,-3.3,-9.8;
move -53,-332,1.1,-17.6,-3.2,-9.8;
move -53,-326.4,1.2,-17.6,-3,-9.8;
move -52,-321.3,1.3,-17.6,-2.9,-9.8;
move -52,-316.5,1.5,-17.6,-2.8,-9.9;
move -51,-312.3,1.6,-17.2,-2.7,-9.9;
move -50,-308.4,1.7,-17.2,-2.6,-9.9;
move -49,-305,1.8,-17.2,-2.4,-9.9;
move -48,-302.1,1.9,-17.2,-2.3,-9.9;
move -47,-299.7,2.1,-16.8,-2.2,-9.9;
move -45,-297.7,2.2,-16.4,-2.1,-9.9;
move -43,-296.2,2.3,-16.4,-1.9,-9.9;
move -41,-295,2.5,-16,-1.8,-9.9;
move -39,-294,2.6,-15.6,-1.7,-9.9;
move -36,-293.3,2.7,-15.2,-1.6,-10;
move -34,-292.9,2.8,-15.2,-1.4,-10;
move -31,-292.6,2.9,-14.4,-1.3,-10;
move -28,-292.6,3.1,-14.4,-1.2,-10;
move -25,-292.6,3.1,-14,-1.1,-10;
move -22,-292.8,3.2,-13.2,-0.9,-10;
move -18,-293,3.3,-12.8,-0.8,-10;
move -15,-293.3,3.4,-12.4,-0.7,-10;
move -11,-293.5,3.4,-11.6,-0.6,-10;
move -8,-293.7,3.5,-11.2,-0.4,-10;
move -4,-293.8,3.6,-10.8,-0.3,-10;
move -1,-293.9,3.7,-10.4,-0.2,-10;
move 3,-293.9,3.7,-10,-0.1,-10;
move 7,-293.7,3.8,-9.6,0.1,-10;
move 11,-293.4,3.9,-8.8,0.2,-10;
move 15,-293,4,-8.4,0.3,-10;
move 19,-292.3,4,-7.6,0.4,-10;
move 23,-291.5,4.1,-7.2,0.6,-10;
move 28,-290.4,4.2,-6.4,0.7,-10;
move 32,-289.2,4.3,-6,0.8,-10;
move 36,-287.8,4.3,-5.2,0.9,-10;
move 41,-286.1,4.4,-4.8,1.1,-10;
move 45,-284.3,4.5,-4,1.2,-10;
move 50,-282.4,4.5,-3.6,1.3,-10;
move 55,-280.3,4.6,-2.8,1.4,-10;
move 60,-278.1,4.7,-2.4,1.6,-10;
move 65,-275.8,4.7,-1.6,1.7,-9.9;
move 70,-273.5,4.8,-0.8,1.8,-9.9;
move 75,-271.2,4.9,-0,1.9,-9.9;
move 80,-268.9,4.9,0.8,2.1,-9.9;
move 86,-266.7,5,1.2,2.2,-9.9;
move 91,-264.7,5.1,2,2.3,-9.9;
move 97,-262.8,5.1,2.8,2.4,-9.9;
move 102,-261.1,5.2,3.6,2.5,-9.9;
move 108,-259.7,5.2,4.4,2.7,-9.9;
move 114,-258.4,5.3,5.2,2.8,-9.8;
move 119,-257.5,5.4,6,2.9,-9.8;
move 125,-256.9,5.4,6.8,3,-9.8;
move 131,-256.6,5.5,7.6,3.2,-9.8;
move 137,-256.6,5.6,8.4,3.3,-9.8;
move 142,-257,5.7,9.2,3.4,-9.7;
move 148,-257.6,5.7,10,3.5,-9.7;
move 154,-258.6,5.8,10.8,3.6,-9.7;
move 159,-259.9,5.9,11.6,3.8,-9.7;
move 164,-261.4,5.9,12.4,3.9,-9.7;
move 170,-263.1,6,12.8,4,-9.6;
move 175,-265.1,6.1,13.6,4.1,-9.6;
move 180,-267.2,6.2,14.4,4.3,-9.6;
move 185,-269.6,6.3,14.8,4.4,-9.5;
move 190,-272.2,6.3,15.6,0,-9.5;
move 195,-274.8,6.4,16.4,0,-9.5;
move 200,-277.6,6.5,17.2,0,-9.5;
move 205,-280.4,6.6,17.6,0,-9.4;
move 210,-283.2,6.6,18.4,0,-9.4;
move 214,-286.1,6.7,19.2,0,-9.4;
move 219,-288.9,6.8,19.6,0,-9.3;
move 223,-291.8,6.8,20.4,0,-9.3;
move 227,-294.7,6.9,20.8,0,-9.3;
move 231,-297.6,7,21.2,0,-9.2;
move 235,-300.4,7.1,22,0,-9.2;
move 239,-303.2,7.2,22.4,0,-9.2;
move 243,-306.1,7.3,22.8,0,-9.1;
move 246,-309,7.4,23.2,0,-9.1;
move 250,-311.9,7.5,24,0,-9;
move 253,-314.9,7.6,24.4,0,-9;
move 256,-317.9,7.7,24.8,0,-9;
move 260,-321.1,7.8,25.2,0,-8.9;
move 262,-324.3,7.9,25.6,0,-8.9;
move 265,-327.6,8,26,0,-8.9;
move 268,-331.1,8.2,26.4,0,-8.8;
move 270,-334.7,8.3,26.8,0,-8.8;
move 273,-338.3,8.4,26.8,0,-8.7;
move 275,-342,8.5,27.2,0,-8.7;
move 277,-345.8,8.6,27.6,0,-8.7;
move 279,-349.5,8.7,28,0,-8.6;
move 281,-353.4,8.8,28,0,-8.6;
move 282,-357.2,9,28.4,0,-8.5;
move 284,-361.1,9.1,28.4,0,-8.5;
move 285,-365,9.2,28.8,0,-8.5;
move 286,-368.9,9.3,28.8,0,-8.4;
move 287,-372.8,9.4,28.8,0,-8.4;
move 288,-376.7,9.5,29.2,0,-8.3;
move 289,-380.7,9.6,29.2,0,-8.3;
move 289,-384.6,9.7,29.2,0,-8.2;
move 290,-388.5,9.8,29.2,0,-8.2;
move 290,-392.4,9.9,29.2,0,-8.1;
move 290,-396.3,9.9,29.2,0,-8.1;
move 290,-400.2,10,29.6,0,-8;
move 290,-404,10.1,29.2,0,-8;
move 290,-407.9,10.2,29.2,0,-7.9;
move 289,-411.7,10.2,29.2,0,-7.9;
move 289,-415.6,10.3,29.2,0,-7.8;
move 288,-419.5,10.4,29.2,0,-7.8;
move 287,-423.4,10.5,28.8,0,-7.7;
move 287,-427.3,10.5,28.8,0,-7.7;
move 286,-431.3,10.6,28.4,0,-7.6;
move 285,-435.3,10.6,28.4,0,-7.6;
move 284,-439.3,10.6,28.4,0,-7.5;
move 283,-443.3,10.7,28.4,0,-7.5;
move 282,-447.3,10.7,28.4,0,-7.4;
move 281,-451.3,10.7,28,0,-7.4;
move 280,-455.3,10.8,28,0,-7.3;
move 279,-459.3,10.8,27.6,0,-7.3;
move 277,-463.2,10.8,27.6,0,-7.2;
move 276,-467.1,10.8,27.2,0,-7.1;
move 274,-470.9,10.8,27.2,10.5,-7.1;
move 273,-474.6,10.7,26.8,10.5,-7;
move 271,-478.2,10.7,26.8,10.6,-7;
move 270,-481.6,10.7,26.4,10.7,-6.9;
move 268,-485,10.7,26.4,10.8,-6.8;
move 266,-488.1,10.7,26,10.9,-6.8;
move 265,-491.1,10.6,25.6,11,-6.7;
move 263,-493.8,10.6,25.6,11.1,-6.7;
move 261,-496.3,10.6,25.2,11.1,-6.6;
move 259,-498.6,10.5,25.2,11.2,-6.5;
move 257,-500.6,10.5,24.8,11.3,-6.5;
move 256,-502.4,10.4,24.4,11.4,-6.4;
move 254,-504,10.3,24.4,11.5,-6.4;
move 252,-505.4,10.3,24,11.6,-6.3;
move 250,-506.5,10.2,23.6,11.6,-6.2;
move 248,-507.5,10.1,23.6,11.7,-6.2;
move 246,-508.2,10,23.2,11.8,-6.1;
move 244,-508.9,9.9,22.8,11.9,-6;
move 242,-509.4,9.8,22.4,11.9,-6;
move 240,-509.8,9.7,22.4,12,-5.9;
move 238,-510.1,9.6,22,12.1,-5.8;
move 236,-510.4,9.5,21.6,12.2,-5.8;
move 234,-510.6,9.4,21.6,12.2,-5.7;
move 233,-510.8,9.3,21.2,12.3,-5.6;
move 231,-511.1,9.2,21.2,12.4,-5.6;
move 230,-511.4,9,20.8,12.5,-5.5;
move 228,-511.9,8.9,20.8,12.5,-5.4;
move 227,-512.5,8.7,20.4,12.6,-5.4;
move 225,-513.2,8.6,20.4,12.7,-5.3;
move 224,-514.2,8.4,20.4,12.7,-5.2;
move 223,-515.4,8.3,20,12.8,-5.1;
move 222,-516.9,8.2,20,12.9,-5.1;
move 220,-518.6,8,19.6,12.9,-5;
move 219,-520.5,7.9,19.6,13,-4.9;
move 218,-522.8,7.7,19.2,13,-4.9;
move 217,-525.2,7.6,19.2,13.1,-4.8;
move 215,-527.9,7.4,19.2,13.2,-4.7;
move 214,-530.7,7.3,18.8,13.2,-4.6;
move 213,-533.7,7.1,18.8,13.3,-4.6;
move 211,-536.9,7,18.4,13.3,-4.5;
move 210,-540.1,6.8,18.4,13.4,-4.4;
move 208,-543.5,6.7,18,13.5,-4.4;
move 207,-546.8,6.5,18,13.5,-4.3;
move 206,-550.2,6.4,17.6,13.6,-4.2;
move 204,-553.5,6.2,17.6,13.6,-4.1;
move 203,-556.7,6.1,17.2,13.7,-4.1;
move 201,-559.8,5.9,17.2,13.7,-4;
move 200,-562.7,5.8,16.8,13.8,-3.9;
move 198,-565.5,5.7,16.8,13.8,-3.8;
move 197,-568.1,5.6,16.4,13.9,-3.8;
move 196,-570.6,5.4,16.4,13.9,-3.7;
move 194,-572.8,5.3,16,14,-3.6;
move 193,-574.9,5.2,16,14,-3.5;
move 192,-576.7,5.1,16,14,-3.4;
move 191,-578.5,5,15.6,14.1,-3.4;
move 189,-580.1,4.9,15.6,14.1,-3.3;
move 188,-581.5,4.8,15.2,14.2,-3.2;
move 187,-582.8,4.7,15.2,14.2,-3.1;
move 185,-584,4.6,15.2,14.3,-3.1;
move 184,-585.1,4.5,14.8,14.3,-3;
move 183,-586.2,4.4,14.8,14.3,-2.9;
move 181,-587.1,4.3,14.4,14.4,-2.8;
move 180,-588.1,4.2,14,14.4,-2.7;
move 178,-588.9,4.1,14,14.4,-2.7;
move 177,-589.8,4.1,13.6,14.5,-2.6;
move 176,-590.6,4,13.6,14.5,-2.5;
move 174,-591.4,3.9,13.6,14.5,-2.4;
move 173,-592.3,3.9,13.2,14.6,-2.3;
move 171,-593.1,3.8,13.2,14.6,-2.3;
move 170,-594,3.8,12.8,14.6,-2.2;
move 168,-594.8,3.7,12.8,14.7,-2.1;
move 167,-595.7,3.7,12.4,14.7,-2;
move 165,-596.6,3.7,12.4,14.7,-1.9;
move 164,-597.5,3.7,12,14.7,-1.9;
move 162,-598.4,3.6,11.6,14.7,-1.8;
move 160,-599.4,3.6,11.6,14.8,-1.7;
move 159,-600.3,3.6,11.2,14.8,-1.6;
move 157,-601.2,3.6,11.2,14.8,-1.5;
move 156,-602.1,3.6,10.8,14.8,-1.5;
move 154,-603,3.6,10.8,14.9,-1.4;
move 153,-603.9,3.6,10.4,14.9,-1.3;
move 152,-604.8,3.6,10.4,14.9,-1.2;
move 150,-605.6,3.7,10,14.9,-1.1;
move 149,-606.4,3.7,10,14.9,-1;
move 148,-607.1,3.7,10,14.9,-1;
move 146,-607.8,3.7,9.6,14.9,-0.9;
move 145,-608.5,3.8,9.6,14.9,-0.8;
move 144,-609.1,3.8,9.2,15,-0.7;
move 143,-609.7,3.8,9.2,15,-0.6;
move 141,-610.3,3.9,8.8,15,-0.5;
move 140,-610.8,3.9,8.8,15,-0.5;
move 139,-611.3,4,8.8,15,-0.4;
move 138,-611.8,4,8.4,15,-0.3;
move 137,-612.3,4.1,8.4,15,-0.2;
move 136,-612.7,4.1,8,15,-0.1;
move 134,-613.2,4.2,8,15,-0;
move 133,-613.7,4.2,8,15,0;
move 132,-614.1,4.3,7.6,15,0.1;
move 131,-614.6,4.4,7.6,15,0.2;
move 130,-615,4.4,7.6,15,0.3;
move 129,-615.5,4.5,7.2,15,0.4;
move 128,-616,4.5,7.2,15,0.5;
move 127,-616.4,4.6,7.2,15,0.5;
move 126,-616.9,4.6,6.8,15,0.6;
move 125,-617.3,4.7,6.8,15,0.7;
move 124,-617.8,4.7,6.8,15,0.8;
move 123,-618.2,4.7,6.4,14.9,0.9;
move 122,-618.6,4.8,6.4,14.9,1;
move 121,-619.1,4.8,6.4,14.9,1;
move 120,-619.5,4.9,6,14.9,1.1;
move 119,-619.9,4.9,6,14.9,1.2;
move 118,-620.3,4.9,6,14.9,1.3;
move 117,-620.7,4.9,5.6,14.9,1.4;
move 116,-621.1,4.9,5.6,14.8,1.4;
move 115,-621.4,5,5.2,14.8,1.5;
move 114,-621.8,5,5.2,14.8,1.6;
move 113,-622.1,5,5.2,14.8,1.7;
move 112,-622.5,5,4.8,14.8,1.8;
move 111,-622.8,5,4.8,14.7,1.9;
move 110,-623.1,5,4.8,14.7,1.9;
move 109,-623.5,5,4.4,14.7,2;
move 108,-623.8,5,4.4,14.7,2.1;
move 108,-624.2,5,4.4,14.6,2.2;
move 107,-624.5,5,4.4,14.6,2.3;
move 106,-624.9,4.9,4,14.6,2.3;
move 106,-625.3,4.9,4,14.6,2.4;
move 105,-625.7,4.9,4,14.5,2.5;
move 105,-626.1,4.9,4,14.5,2.6;
move 104,-626.5,4.8,4,14.5,2.7;
move 103,-627,4.8,4,14.4,2.7;
move 103,-627.4,4.8,3.6,14.4,2.8;
move 102,-627.8,4.7,3.6,14.4,2.9;
move 101,-628.3,4.7,3.6,14.3,3;
move 101,-628.7,4.6,3.6,14.3,3.1;
move 100,-629.1,4.6,3.2,14.3,3.1;
move 99,-629.6,4.5,3.2,14.2,3.2;
move 99,-630,4.4,3.2,14.2,3.3;
move 98,-630.4,4.4,3.2,14.1,3.4;
move 97,-630.7,4.3,2.8,14.1,3.4;
move 96,-631.1,4.2,2.8,14,3.5;
move 96,-631.4,4.1,2.8,14,3.6;
move 95,-631.7,4,2.8,14,3.7;
move 94,-632,4,2.4,13.9,3.7;
move 94,-632.3,3.9,2.4,13.9,3.8;
move 93,-632.5,3.8,2.4,13.8,3.9;
move 92,-632.7,3.7,2.4,13.8,4;
move 92,-632.9,3.6,2.4,13.7,4;
move 91,-633,3.5,2,13.7,4.1;
move 90,-633.1,3.4,2,13.6,4.2;
move 90,-633.2,3.3,2,13.6,4.3;
move 89,-633.3,3.2,2,13.5,4.3;
move 88,-633.4,3.1,1.6,13.4,4.4;
move 88,-633.5,3,1.6,13.4,4.5;
move 87,-633.5,2.9,1.6,13.3,4.6;
move 86,-633.6,2.8,1.6,13.3,4.6;
move 86,-633.6,2.8,1.2,13.2,4.7;
move 85,-633.6,2.7,1.2,13.2,4.8;
move 84,-633.7,2.6,1.2,13.1,4.9;
move 84,-633.7,2.6,1.2,13,4.9;
move 83,-633.7,2.5,1.2,13,5;
move 83,-633.7,2.4,0.8,12.9,5.1;
move 82,-633.7,2.4,0.8,12.8,5.1;
move 82,-633.7,2.3,0.8,12.8,5.2;
move 81,-633.7,2.2,0.8,12.7,5.3;
move 81,-633.7,2.2,0.8,12.7,5.4;
move 80,-633.7,2.1,0.8,12.6,5.4;
move 80,-633.7,2.1,0.4,12.5,5.5;
move 79,-633.7,2,0.4,12.4,5.6;
move 79,-633.7,2,0.4,12.4,5.6;
move 78,-633.7,1.9,0.4,12.3,5.7;
move 77,-633.7,1.9,0.4,12.2,5.8;
move 77,-633.7,1.8,0.4,12.2,5.8;
move 76,-633.7,1.8,0,12.1,5.9;
move 76,-633.7,1.8,-0,12,6;
move 75,-633.7,1.7,-0,11.9,6;
move 74,-633.7,1.7,-0,11.9,6.1;
move 74,-633.7,1.7,-0.4,11.8,6.2;
move 73,-633.7,1.7,-0.4,11.7,6.2;
move 73,-633.7,1.7,-0.4,11.6,6.3;
move 72,-633.7,1.6,-0.4,11.5,6.3;
move 72,-633.7,1.6,-0.4,11.5,6.4;
move 71,-633.7,1.6,-0.4,11.4,6.5;
move 71,-633.7,1.6,-0.8,11.3,6.5;
move 70,-633.7,1.6,-0.8,11.2,6.6;
move 70,-633.7,1.6,-0.8,11.1,6.7;
move 70,-633.6,1.6,-0.8,11.1,6.7;
move 69,-633.6,1.6,-0.8,11,6.8;
move 69,-633.6,1.7,-0.8,10.9,6.8;
move 69,-633.5,1.7,-0.8,10.8,6.9;
move 68,-633.4,1.7,-0.8,10.7,7;
move 68,-633.4,1.7,-1.2,10.6,7;
move 67,-633.3,1.7,-1.2,10.5,7.1;
move 67,-633.2,1.7,-1.2,10.4,7.1;
move 67,-633,1.7,-1.2,10.4,7.2;
move 66,-632.9,1.8,-1.2,10.3,7.2;
move 66,-632.7,1.8,-1.2,10.2,7.3;
move 66,-632.5,1.9,-1.2,10.1,7.4;
move 65,-632.3,1.9,-1.2,10,7.4;
move 65,-632,1.9,-1.6,9.9,7.5;
move 65,-631.7,2,-1.6,9.8,7.5;
move 64,-631.4,2,-1.6,9.7,7.6;
move 64,-631.1,2.1,-1.6,9.6,7.6;
move 64,-630.8,2.1,-1.6,9.5,7.7;
move 64,-630.4,2.2,-1.6,9.4,7.7;
move 63,-630,2.2,-1.6,9.3,7.8;
move 63,-629.6,2.3,-1.6,9.2,7.8;
move 63,-629.2,2.3,-1.6,9.1,7.9;
move 63,-628.7,2.4,-1.6,9,7.9;
move 62,-628.3,2.5,-1.6,8.9,8;
move 62,-627.9,2.5,-2,8.8,8;
move 62,-627.4,2.6,-2,8.7,8.1;
move 61,-627,2.6,-2,8.6,8.1;
move 61,-626.6,2.7,-2,8.5,8.2;
move 61,-626.2,2.8,-2,8.4,8.2;
move 61,-625.9,2.8,-2,8.3,8.3;
move 61,-625.6,2.9,-2,8.2,8.3;
move 61,-625.3,2.9,-2,8.1,8.4;
move 61,-625.1,3,-2,8,8.4;
move 61,-624.9,3.1,-2,7.9,8.4;
move 61,-624.7,3.1,-2,7.8,8.5;
move 61,-624.6,3.2,-2,7.7,8.5;
move 60,-624.5,3.2,-2,7.6,8.6;
move 60,-624.5,3.3,-2,7.5,8.6;
move 60,-624.5,3.3,-2,7.3,8.7;
move 60,-624.5,3.4,-2,7.2,8.7;
move 60,-624.6,3.5,-2,7.1,8.7;
move 59,-624.7,3.5,-2,7,8.8;
move 59,-624.9,3.5,-2.4,6.9,8.8;
move 59,-625,3.6,-2.4,6.8,8.9;
move 58,-625.2,3.6,-2.4,6.7,8.9;
move 58,-625.4,3.7,-2.4,6.6,8.9;
move 58,-625.6,3.7,-2.4,6.5,9;
move 57,-625.8,3.8,-2.4,6.3,9;
move 57,-626,3.8,-2.4,6.2,9;
move 56,-626.2,3.8,-2.4,6.1,9.1;
move 56,-626.4,3.9,-2.8,6,9.1;
move 56,-626.6,3.9,-2.8,5.9,9.2;
move 55,-626.8,4,-2.8,5.8,9.2;
move 55,-626.9,4,-2.8,5.7,9.2;
move 55,-626.9,4.1,-2.8,5.5,9.3;
move 54,-626.9,4.1,-2.8,5.4,9.3;
move 54,-626.9,4.1,-2.8,5.3,9.3;
move 54,-626.9,4.2,-2.8,5.2,9.4;
move 53,-626.8,4.2,-2.8,5.1,9.4;
move 53,-626.6,4.2,-3.2,5,9.4;
move 53,-626.4,4.3,-3.2,4.8,9.4;
move 52,-626.1,4.3,-3.2,4.7,9.5;
move 52,-625.8,4.3,-3.2,4.6,9.5;
move 52,-625.4,4.3,-3.2,4.5,9.5;
move 51,-625,4.4,-3.2,4.4,9.6;
move 51,-624.6,4.4,-3.2,4.2,9.6;
move 51,-624.2,4.4,-3.2,4.1,9.6;
move 50,-623.7,4.4,-3.6,4,9.6;
move 50,-623.2,4.4,-3.6,3.9,9.7;
move 50,-622.7,4.4,-3.6,3.8,9.7;
move 49,-622.2,4.5,-3.6,3.6,9.7;
move 49,-621.7,4.5,-3.6,3.5,9.7;
move 49,-621.1,4.5,-3.6,3.4,9.8;
move 48,-620.6,4.5,-3.6,3.3,9.8;
move 48,-620,4.5,-3.6,3.2,9.8;
move 48,-619.5,4.5,-3.6,3,9.8;
move 47,-618.9,4.5,-3.6,2.9,9.8;
move 47,-618.3,4.6,-4,2.8,9.9;
move 46,-617.7,4.6,-4,2.7,9.9;
move 46,-617.1,4.6,-4,2.5,9.9;
move 45,-616.5,4.6,-4,2.4,9.9;
move 45,-615.9,4.7,-4,2.3,9.9;
move 44,-615.3,4.7,-4.4,2.2,9.9;
move 43,-614.8,4.7,-4.4,2,9.9;
move 43,-614.2,4.7,-4.4,1.9,9.9;
move 42,-613.7,4.7,-4.4,1.8,9.9;
move 41,-613.2,4.8,-4.8,1.7,9.9;
move 41,-612.6,4.8,-4.8,1.5,10;
move 40,-612.2,4.8,-4.8,1.4,10;
move 39,-611.7,4.8,-4.8,1.3,10;
move 39,-611.3,4.8,-5.2,1.2,10;
move 38,-610.9,4.9,-5.2,1,10;
move 38,-610.6,4.9,-5.2,0.9,10;
move 37,-610.2,4.9,-5.2,0.8,10;
move 37,-609.9,5,-5.2,0.7,10;
move 36,-609.6,5,-5.2,0.5,10;
move 35,-609.3,5,-5.2,0.4,10;
move 35,-609,5,-5.6,0.3,10;
move 34,-608.8,5.1,-5.6,0.2,10;
move 33,-608.5,5.1,-5.6,0,10;
move 32,-608.3,5.1,-6,-0.1,10;
move 31,-608,5.1,-6,-0.2,10;
move 31,-607.7,5.2,-6,-0.3,10;
move 30,-607.5,5.2,-6,-0.5,10;
move 29,-607.2,5.3,-6.4,-0.6,10;
move 28,-606.9,5.3,-6.4,-0.7,10;
move 27,-606.5,5.3,-6.8,-0.8,10;
move 26,-606.2,5.4,-6.8,-1,10;
move 25,-605.8,5.4,-6.8,-1.1,10;
move 24,-605.4,5.4,-7.2,-1.2,10;
move 23,-605,5.5,-7.2,-1.3,10;
move 21,-604.6,5.5,-7.2,-1.4,10;
move 20,-604.1,5.5,-7.6,-1.6,9.9;
move 19,-603.6,5.6,-7.6,-1.7,9.9;
move 18,-603.1,5.6,-7.6,-1.8,9.9;
move 17,-602.6,5.7,-8,-1.9,9.9;
move 16,-602.1,5.7,-8,-2.1,9.9;
move 15,-601.6,5.8,-8,-2.2,9.9;
move 14,-601.1,5.8,-8.4,-2.3,9.9;
move 13,-600.6,5.8,-8.4,-2.4,9.9;
move 12,-600.1,5.9,-8.8,-2.6,9.9;
move 11,-599.6,5.9,-8.8,-2.7,9.8;
move 9,-599.2,5.9,-8.8,-2.8,9.8;
move 8,-598.8,6,-9.2,-2.9,9.8;
move 7,-598.4,6,-9.2,-3.1,9.8;
move 6,-598,6,-9.6,-3.2,9.8;
move 5,-597.7,6.1,-9.6,-3.3,9.7;
move 4,-597.4,6.2,-10,-3.4,9.7;
move 3,-597.2,6.2,-10,-3.5,9.7;
move 1,-596.9,6.3,-10,-3.7,9.7;
move 0,-596.7,6.3,-10,-3.8,9.7;
move -1,-596.5,6.4,-10.4,-3.9,9.6;
move -2,-596.2,6.4,-10.4,-4,9.6;
move -3,-596,6.5,-10.8,-4.1,9.6;
move -4,-595.7,6.5,-10.8,-4.3,9.5;
move -5,-595.4,6.6,-10.8,-4.4,9.5;
move -6,-595,6.6,-11.2,-4.5,9.5;
move -7,-594.6,6.7,-11.2,-4.6,9.5;
move -7,-594.1,6.7,-11.2,-4.7,9.4;
move -8,-593.5,6.8,-11.6,-4.9,9.4;
move -9,-592.8,6.8,-11.6,-5,9.4;
move -9,-591.9,6.9,-11.6,-5.1,9.3;
move -10,-591,6.9,-11.6,-5.2,9.3;
move -10,-589.9,6.9,-11.6,-5.3,9.3;
move -10,-588.7,7,-11.6,-5.4,9.2;
move -11,-587.4,7,-12,-5.6,9.2;
move -11,-585.9,7.1,-12,-5.7,9.2;
move -11,-584.2,7.1,-12,-5.8,9.1;
move -11,-582.3,7.1,-11.6,-5.9,9.1;
move -10,-580.3,7.2,-11.6,-6,9.1;
move -10,-578.1,7.2,-11.6,-6.1,9;
move -10,-575.7,7.2,-11.6,-6.3,9;
move -9,-573.2,7.3,-11.6,-6.4,9;
move -9,-570.6,7.3,-11.6,-6.5,8.9;
move -8,-567.8,7.3,-11.6,-6.6,8.9;
move -7,-565,7.3,-11.2,-6.7,8.8;
move -6,-562.1,7.4,-11.2,-6.8,8.8;
move -5,-559.1,7.4,-11.2,-6.9,8.8;
move -4,-556.1,7.4,-10.8,-7,8.7;
move -3,-553.1,7.4,-10.8,-7.2,8.7;
move -1,-550,7.4,-10.4,-7.3,8.7;
move 0,-547.1,7.4,-10.4,-7.4,8.6;
move 2,-544.1,7.4,-10,-7.5,8.6;
move 3,-541.2,7.4,-10,-7.6,8.5;
move 5,-538.4,7.4,-9.6,-7.7,8.5;
move 7,-535.7,7.4,-9.2,-7.8,8.4;
move 9,-533,7.4,-9.2,-7.9,8.4;
move 11,-530.5,7.4,-8.8,-8,8.4;
move 13,-528,7.4,-8.4,-8.1,8.3;
move 16,-525.7,7.3,-8.4,-8.2,8.3;
move 18,-523.4,7.3,-8,-8.3,8.2;
move 20,-521.3,7.3,-7.6,-8.4,8.2;
move 23,-519.2,7.3,-7.2,-8.5,8.1;
move 26,-517.3,7.2,-6.8,-8.6,8.1;
move 28,-515.5,7.2,-6.4,-8.7,8;
move 31,-513.9,7.2,-6,-8.8,8;
move 34,-512.3,7.2,-5.6,-8.9,7.9;
move 37,-510.9,7.1,-5.2,-9,7.9;
move 40,-509.7,7.1,-4.8,-9.1,7.8;
move 43,-508.7,7,-4.4,-9.2,7.8;
move 46,-507.8,7,-4,-9.3,7.7;
move 49,-507.1,6.9,-3.6,-9.4,7.7;
move 52,-506.6,6.9,-3.2,-9.5,7.6;
move 55,-506.2,6.8,-2.8,-9.6,7.6;
move 58,-506.1,6.7,-2.4,-9.7,7.5;
move 61,-506.1,6.6,-2,-9.8,7.5;
move 63,-506.3,6.6,-1.6,-9.9,7.4;
move 66,-506.6,6.5,-1.2,-10,7.4;
move 69,-507.1,6.4,-0.8,-10.1,7.3;
move 72,-507.7,6.4,-0.4,-10.2,7.3;
move 75,-508.4,6.3,-0,-10.3,7.2;
move 78,-509.2,6.2,0.4,-10.4,7.1;
move 81,-510,6.1,0.8,-10.5,7.1;
move 83,-511,6,1.2,-10.6,7;
move 86,-512,5.9,1.6,-10.6,7;
move 88,-513,5.9,2,-10.7,6.9;
move 91,-514.1,5.8,2,-10.8,6.8;
move 93,-515.2,5.7,2.4,-10.9,6.8;
move 96,-516.4,5.6,2.8,-11,6.7;
move 98,-517.5,5.5,3.2,-11.1,6.7;
move 100,-518.7,5.4,3.6,-11.2,6.6;
move 102,-519.8,5.3,3.6,-11.2,6.5;
move 104,-521,5.2,4,-11.3,6.5;
move 106,-522.1,5.1,4.4,-11.4,6.4;
move 108,-523.2,5,4.4,-11.5,6.4;
move 109,-524.2,4.9,4.8,-11.6,6.3;
move 111,-525.3,4.8,4.8,-11.6,6.2;
move 112,-526.4,4.8,5.2,-11.7,6.2;
move 114,-527.5,4.7,5.2,-11.8,6.1;
move 115,-528.7,4.6,5.6,-11.9,6;
move 116,-529.8,4.5,5.6,-12,6;
move 117,-530.9,4.4,6,-12,5.9;
move 118,-532.1,4.4,6,-12.1,5.8;
move 119,-533.4,4.3,6,-12.2,5.8;
move 120,-534.6,4.2,6,-12.2,5.7;
move 120,-535.9,4.1,6.4,-12.3,5.6;
move 121,-537.3,4,6.4,-12.4,5.6;
move 121,-538.7,4,6.4,-12.5,5.5;
move 121,-540.2,3.9,6.4,-12.5,5.4;
move 121,-541.7,3.8,6.4,-12.6,5.4;
move 121,-543.2,3.8,6.4,-12.7,5.3;
move 121,-544.8,3.7,6.4,-12.7,5.2;
move 121,-546.4,3.6,6.4,-12.8,5.1;
move 120,-548.1,3.6,6,-12.9,5.1;
move 120,-549.7,3.5,6,-12.9,5;
move 119,-551.3,3.4,6,-13,4.9;
move 119,-552.9,3.4,6,-13.1,4.9;
move 118,-554.5,3.3,6,-13.1,4.8;
move 117,-556,3.2,5.6,-13.2,4.7;
move 117,-557.5,3.1,5.6,-13.2,4.6;
move 116,-558.9,3.1,5.6,-13.3,4.6;
move 115,-560.2,3,5.6,-13.3,4.5;
move 114,-561.4,3,5.2,-13.4,4.4;
move 113,-562.5,2.9,5.2,-13.5,4.4;
move 112,-563.5,2.8,5.2,-13.5,4.3;
move 111,-564.4,2.8,4.8,-13.6,4.2;
move 110,-565.2,2.7,4.8,-13.6,4.1;
move 109,-565.8,2.6,4.8,-13.7,4.1;
move 108,-566.3,2.6,4.4,-13.7,4;
move 106,-566.7,2.5,4.4,-13.8,3.9;
move 105,-566.9,2.5,4,-13.8,3.8;
move 103,-567,2.4,4,-13.9,3.8;
move 102,-567,2.4,3.6,-13.9,3.7;
move 101,-566.8,2.3,3.2,-14,3.6;
move 99,-566.5,2.3,3.2,-14,3.5;
move 98,-566.1,2.2,2.8,-14.1,3.4;
move 96,-565.6,2.2,2.8,-14.1,3.4;
move 95,-564.9,2.2,2.8,-14.1,3.3;
move 94,-564.2,2.1,2.4,-14.2,3.2;
move 93,-563.4,2.1,2.4,-14.2,3.1;
move 91,-562.6,2,2,-14.3,3.1;
move 90,-561.7,2,2,-14.3,3;
move 89,-560.8,1.9,2,-14.3,2.9;
move 88,-559.8,1.9,1.6,-14.4,2.8;
move 87,-558.8,1.9,1.6,-14.4,2.7;
move 86,-557.9,1.8,1.2,-14.4,2.7;
move 85,-556.9,1.8,1.2,-14.5,2.6;
move 84,-555.9,1.8,1.2,-14.5,2.5;
move 83,-554.9,1.7,1.2,-14.5,2.4;
move 81,-554,1.7,0.8,-14.6,2.3;
move 80,-553.1,1.7,0.8,-14.6,2.3;
move 79,-552.2,1.6,0.4,-14.6,2.2;
move 78,-551.4,1.6,0.4,-14.7,2.1;
move 78,-550.7,1.6,0,-14.7,2;
move 77,-550,1.6,0,-14.7,1.9;
move 76,-549.4,1.5,0,-14.7,1.9;
move 75,-548.8,1.5,0,-14.8,1.8;
move 75,-548.4,1.5,-0,-14.8,1.7;
move 74,-547.9,1.5,-0.4,-14.8,1.6;
move 74,-547.6,1.4,-0.4,-14.8,1.5;
move 73,-547.3,1.4,-0.4,-14.8,1.5;
move 73,-547.1,1.4,-0.4,-14.9,1.4;
move 73,-546.9,1.4,-0.4,-14.9,1.3;
move 72,-546.8,1.4,-0.4,-14.9,1.2;
move 72,-546.7,1.4,-0.4,-14.9,1.1;
move 72,-546.8,1.4,-0.4,-14.9,1;
move 72,-546.8,1.3,-0.4,-14.9,1;
move 71,-547,1.3,-0.4,-14.9,0.9;
move 71,-547.1,1.3,-0.4,-14.9,0.8;
move 71,-547.3,1.3,-0.8,-15,0.7;
move 71,-547.6,1.3,-0.8,-15,0.6;
move 70,-547.8,1.3,-0.8,-15,0.5;
move 70,-548.1,1.3,-0.8,-15,0.5;
move 70,-548.4,1.3,-0.8,-15,0.4;
move 70,-548.8,1.4,-0.8,-15,0.3;
move 70,-549.1,1.4,-0.8,-15,0.2;
move 70,-549.5,1.4,-0.4,-15,0.1;
move 70,-549.8,1.4,-0.8,-15,0;
move 71,-550.2,1.5,-0.8,-15,-0;
move 71,-550.5,1.5,-0.4,-15,-0.1;
move 71,-550.8,1.5,-0.4,-15,-0.2;
move 71,-551.1,1.6,-0.4,-15,-0.3;
move 71,-551.4,1.6,-0.8,-15,-0.4;
move 70,-551.7,1.7,-0.8,-15,-0.5;
move 70,-552,1.7,-0.8,-15,-0.5;
move 70,-552.2,1.7,-0.8,-15,-0.6;
move 70,-552.4,1.8,-0.8,-15,-0.7;
move 70,-552.6,1.8,-0.4,-15,-0.8;
move 70,-552.8,1.9,-0.8,-14.9,-0.9;
move 70,-552.9,2,-0.8,-14.9,-1;
move 71,-553,2,-0.8,-14.9,-1;
move 71,-553.1,2.1,-0.4,-14.9,-1.1;
move 70,-553.2,2.1,-0.4,-14.9,-1.2;
move 70,-553.3,2.2,-0.4,-14.9,-1.3;
move 70,-553.4,2.2,-0.8,-14.9,-1.4;
move 70,-553.4,2.3,-0.8,-14.8,-1.4;
move 70,-553.5,2.4,-0.8,-14.8,-1.5;
move 70,-553.5,2.5,-0.8,-14.8,-1.6;
move 70,-553.6,2.5,-0.8,-14.8,-1.7;
move 70,-553.6,2.6,-0.8,-14.8,-1.8;
move 70,-553.7,2.7,-0.8,-14.7,-1.9;
move 70,-553.7,2.8,-0.8,-14.7,-1.9;
move 70,-553.7,2.9,-0.8,-14.7,-2;
move 69,-553.7,3,-0.8,-14.7,-2.1;
move 69,-553.7,3.1,-0.8,-14.6,-2.2;
move 69,-553.7,3.2,-0.8,-14.6,-2.3;
move 69,-553.7,3.3,-0.8,-14.6,-2.3;
move 69,-553.7,3.4,-0.8,-14.6,-2.4;
move 69,-553.7,3.5,-0.8,-14.5,-2.5;
move 69,-553.7,3.6,-0.8,-14.5,-2.6;
move 69,-553.6,3.7,-0.8,-14.5,-2.7;
move 69,-553.6,3.8,-0.8,-14.4,-2.7;
move 69,-553.6,3.9,-0.8,-14.4,-2.8;
move 69,-553.5,4,-0.8,-14.4,-2.9;
move 69,-553.5,4.2,-0.8,-14.3,-3;
move 69,-553.4,4.3,-0.8,-14.3,-3.1;
move 69,-553.3,4.4,-0.8,-14.2,-3.1;
move 69,-553.1,4.5,-0.8,-14.2,-3.2;
move 70,-553,4.6,-0.8,-14.2,-3.3;
move 70,-552.8,4.7,-0.8,-14.1,-3.4;
move 70,-552.5,4.8,-0.8,-14.1,-3.4;
move 70,-552.3,5,-0.8,-14,-3.5;
move 70,-552,5.1,-0.8,-14,-3.6;
move 70,-551.7,5.2,-0.8,-13.9,-3.7;
move 70,-551.4,5.4,-0.8,-13.9,-3.7;
move 71,-551,5.5,-0.8,-13.9,-3.8;
move 71,-550.6,5.6,-0.4,-13.8,-3.9;
move 71,-550.2,5.7,-0.4,-13.8,-4;
move 72,-549.8,5.9,-0.4,-13.7,-4;
move 72,-549.3,6,-0.4,-13.7,-4.1;
move 72,-548.9,6.1,-0.4,-13.6,-4.2;
move 72,-548.4,6.2,-0.4,-13.6,-4.3;
move 72,-547.9,6.4,-0.4,-13.5,-4.3;
move 73,-547.4,6.5,-0.4,-13.4,-4.4;
move 73,-546.9,6.6,-0.4,-13.4,-4.5;
move 73,-546.4,6.8,-0.4,-13.3,-4.6;
move 73,-545.9,6.9,-0.4,-13.3,-4.6;
move 73,-545.5,7,-0.4,-13.2,-4.7;
move 73,-545.1,7.1,-0,-13.2,-4.8;
move 74,-544.7,7.2,-0,-13.1,-4.9;
move 74,-544.3,7.3,-0.4,-13,-4.9;
move 74,-544,7.4,-0.4,-13,-5;
move 74,-543.7,7.5,-0.4,-12.9,-5.1;
move 74,-543.4,7.6,-0,-12.8,-5.1;
move 75,-543.3,7.7,-0,-12.8,-5.2;
move 75,-543.1,7.9,0,-12.7,-5.3;
move 75,-543.1,8,0,-12.6,-5.4;
move 75,-543.1,8.1,-0,-12.6,-5.4;
move 75,-543.2,8.2,0,-12.5,-5.5;
move 75,-543.3,8.3,0,-12.4,-5.6;
move 75,-543.6,8.3,0,-12.4,-5.6;
move 75,-543.9,8.4,0,-12.3,-5.7;
move 75,-544.3,8.5,0,-12.2,-5.8;
move 75,-544.8,8.6,0,-12.1,-5.8;
move 75,-545.3,8.6,0,-12.1,-5.9;
move 75,-545.9,8.7,0,-12,-6;
move 75,-546.5,8.8,0,-11.9,-6;
move 75,-547.2,8.8,0,-11.8,-6.1;
move 75,-547.9,8.8,0,-11.8,-6.2;
move 75,-548.7,8.9,0,-11.7,-6.2;
move 75,-549.4,8.9,0,-11.6,-6.3;
move 75,-550.2,9,-0,-11.5,-6.3;
move 75,-550.9,9,-0,-11.5,-6.4;
move 75,-551.6,9,-0,-11.4,-6.5;
move 74,-552.3,9.1,-0,-11.3,-6.5;
move 74,-553,9.1,-0,-11.2,-6.6;
move 74,-553.6,9.1,-0,-11.1,-6.7;
move 73,-554.2,9.1,-0.4,-11,-6.7;
move 73,-554.7,9.1,-0.4,-11,-6.8;
move 72,-555.2,9.1,-0.4,-10.9,-6.8;
move 71,-555.6,9.2,-0.4,-10.8,-6.9;
move 70,-556,9.1,-0.8,-10.7,-7;
move 70,-556.3,9.1,-0.8,-10.6,-7;
move 69,-556.5,9.1,-0.8,-10.5,-7.1;
move 68,-556.7,9.1,-0.8,-10.4,-7.1;
move 67,-556.9,9.1,-1.2,-10.3,-7.2;
move 66,-557,9.1,-1.2,-10.3,-7.2;
move 65,-557.1,9,-1.6,-10.2,-7.3;
move 64,-557.1,9,-1.6,-10.1,-7.4;
move 63,-557.2,8.9,-1.6,-10,-7.4;
move 62,-557.2,8.9,-2,-9.9,-7.5;
move 60,-557.2,8.8,-2,-9.8,-7.5;
move 59,-557.2,8.8,-2,-9.7,-7.6;
move 58,-557.2,8.7,-2.4,-9.6,-7.6;
move 57,-557.2,8.7,-2.4,-9.5,-7.7;
move 55,-557.2,8.6,-2.8,-9.4,-7.7;
move 54,-557.2,8.5,-2.8,-9.3,-7.8;
move 53,-557.3,8.5,-3.2,-9.2,-7.8;
move 52,-557.4,8.4,-3.2,-9.1,-7.9;
move 50,-557.5,8.3,-3.6,-9,-7.9;
move 49,-557.7,8.2,-3.6,-8.9,-8;
move 48,-557.8,8.1,-3.6,-8.8,-8;
move 46,-557.9,8.1,-4,-8.7,-8.1;
move 45,-558.1,8,-4,-8.6,-8.1;
move 43,-558.2,7.9,-4.4,-8.5,-8.2;
move 42,-558.3,7.8,-4.4,-8.4,-8.2;
move 40,-558.4,7.8,-4.8,-8.3,-8.3;
move 39,-558.4,7.7,-5.2,-8.2,-8.3;
move 38,-558.4,7.6,-5.2,-8.1,-8.4;
move 36,-558.3,7.6,-5.2,-8,-8.4;
move 35,-558.1,7.5,-5.6,-7.9,-8.4;
move 33,-557.9,7.4,-5.6,-7.8,-8.5;
move 32,-557.5,7.4,-6,-7.7,-8.5;
move 30,-557.1,7.3,-6,-7.5,-8.6;
move 29,-556.5,7.2,-6.4,-7.4,-8.6;
move 28,-555.8,7.2,-6.4,-7.3,-8.7;
move 26,-555,7.1,-6.8,-7.2,-8.7;
move 25,-554.1,7,-6.8,-7.1,-8.7;
move 24,-553.1,6.9,-7.2,-7,-8.8;
move 22,-552,6.9,-7.2,-6.9,-8.8;
move 21,-550.8,6.8,-7.6,-6.8,-8.9;
move 20,-549.5,6.8,-7.6,-6.7,-8.9;
move 19,-548.1,6.7,-7.6,-6.6,-8.9;
move 18,-546.6,6.7,-8,-6.4,-9;
move 17,-545.1,6.6,-8,-6.3,-9;
move 16,-543.5,6.6,-8,-6.2,-9;
move 15,-541.8,6.5,-8,-6.1,-9.1;
move 15,-540.2,6.5,-8.4,-6,-9.1;
move 14,-538.5,6.4,-8.4,-5.9,-9.2;
move 13,-536.8,6.4,-8.4,-5.8,-9.2;
move 13,-535,6.3,-8.8,-5.6,-9.2;
move 12,-533.3,6.3,-8.8,-5.5,-9.3;
move 11,-531.6,6.2,-8.8,-5.4,-9.3;
move 11,-529.9,6.2,-8.8,-5.3,-9.3;
move 11,-528.2,6.2,-8.8,-5.2,-9.4;
move 10,-526.6,6.2,-8.8,-5.1,-9.4;
move 10,-524.9,6.1,-8.8,-4.9,-9.4;
move 9,-523.3,6.1,-8.8,-4.8,-9.4;
move 9,-521.7,6.1,-9.2,-4.7,-9.5;
move 9,-520.1,6.1,-9.2,-4.6,-9.5;
move 8,-518.6,6.1,-9.2,-4.5,-9.5;
move 8,-517,6.2,-9.2,-4.3,-9.6;
move 8,-515.6,6.2,-9.2,-4.2,-9.6;
move 8,-514.1,6.2,-9.2,-4.1,-9.6;
move 8,-512.7,6.2,-9.2,-4,-9.6;
move 8,-511.4,6.3,-9.2,-3.9,-9.7;
move 8,-510,6.3,-9.2,-3.7,-9.7;
move 8,-508.7,6.3,-9.2,-3.6,-9.7;
move 8,-507.4,6.3,-9.2,-3.5,-9.7;
move 8,-506.2,6.4,-9.2,-3.4,-9.8;
move 8,-505.1,6.4,-9.2,-3.3,-9.8;
move 8,-504,6.5,-9.2,-3.1,-9.8;
move 8,-503,6.5,-9.2,-3,-9.8;
move 8,-502.1,6.6,-9.2,-2.9,-9.8;
move 8,-501.3,6.7,-9.2,-2.8,-9.9;
move 7,-500.6,6.7,-9.2,-2.6,-9.9;
move 7,-499.9,6.8,-9.2,-2.5,-9.9;
move 7,-499.3,6.8,-9.2,-2.4,-9.9;
move 7,-498.8,6.9,-9.2,-2.3,-9.9;
move 7,-498.5,6.9,-9.2,-2.2,-9.9;
move 6,-498.2,7,-9.2,-2,-9.9;
move 6,-498,7.1,-9.6,-1.9,-9.9;
move 5,-497.9,7.1,-9.6,-1.8,-9.9;
move 5,-497.9,7.2,-9.6,-1.7,-9.9;
move 4,-498,7.3,-9.6,-1.5,-10;
move 4,-498.2,7.4,-9.6,-1.4,-10;
move 3,-498.4,7.5,-10,-1.3,-10;
move 2,-498.7,7.6,-10,-1.2,-10;
move 2,-499.1,7.6,-10,-1,-10;
move 1,-499.5,7.7,-10,-0.9,-10;
move 0,-499.9,7.8,-10,-0.8,-10;
move 0,-500.3,7.9,-10,-0.7,-10;
move -1,-500.8,8,-10.4,-0.5,-10;
move -2,-501.2,8,-10.4,-0.4,-10;
move -4,-501.5,8.1,-10.8,-0.3,-10;
move -5,-501.9,8.2,-10.8,-0.2,-10;
move -6,-502.1,8.3,-11.2,-0,-10;
move -7,-502.3,8.4,-11.2,0.1,-10;
move -9,-502.3,8.4,-11.2,0.2,-10;
move -10,-502.3,8.5,-11.6,0.3,-10;
move -12,-502.2,8.6,-12,0.5,-10;
move -13,-502,8.7,-12,0.6,-10;
move -15,-501.8,8.7,-12.4,0.7,-10;
move -17,-501.4,8.8,-12.4,0.8,-10;
move -18,-500.9,8.8,-12.8,1,-10;
move -20,-500.3,8.9,-12.8,1.1,-10;
move -22,-499.6,8.9,-13.2,1.2,-10;
move -24,-498.9,9,-13.6,1.3,-10;
move -25,-498.1,9,-13.6,1.5,-10;
move -27,-497.2,9.1,-14,1.6,-9.9;
move -29,-496.2,9.1,-14,1.7,-9.9;
move -31,-495.1,9.1,-14.4,1.8,-9.9;
move -33,-494,9.2,-14.8,2,-9.9;
move -35,-492.7,9.2,-14.8,2.1,-9.9;
move -37,-491.5,9.2,-15.2,2.2,-9.9;
move -39,-490.2,9.2,-15.6,2.3,-9.9;
move -41,-488.8,9.2,-16,2.5,-9.9;
move -43,-487.3,9.2,-16,2.6,-9.9;
move -45,-485.8,9.3,-16.4,2.7,-9.8;
move -47,-484.3,9.3,-16.8,2.8,-9.8;
move -48,-482.7,9.3,-16.8,2.9,-9.8;
move -50,-481.1,9.2,-17.2,3.1,-9.8;
move -52,-479.3,9.2,-17.2,3.2,-9.8;
move -54,-477.6,9.2,-17.6,3.3,-9.7;
move -56,-475.7,9.2,-18,3.4,-9.7;
move -57,-473.8,9.2,-18,3.6,-9.7;
move -59,-471.8,9.2,-18.4,3.7,-9.7;
move -61,-469.8,9.1,-18.4,3.8,-9.7;
move -63,-467.7,9.1,-18.8,3.9,-9.6;
move -64,-465.6,9.1,-19.2,4,-9.6;
move -66,-463.4,9,-19.2,4.2,-9.6;
move -67,-461.1,9,-19.6,4.3,-9.5;
move -69,-458.8,9,-19.6,4.4,-9.5;
move -70,-456.5,8.9,-20,4.5,-9.5;
move -71,-454.1,8.8,-20,4.6,-9.5;
move -72,-451.6,8.8,-20,4.8,-9.4;
move -74,-449.1,8.7,-20.4,4.9,-9.4;
move -75,-446.5,8.6,-20.4,5,-9.4;
move -76,-443.9,8.6,-20.8,5.1,-9.3;
move -76,-441.3,8.5,-20.8,5.2,-9.3;
move -77,-438.7,8.4,-20.8,5.3,-9.3;
move -78,-436.1,8.3,-20.8,5.5,-9.2;
move -79,-433.5,8.2,-20.8,5.6,-9.2;
move -79,-430.8,8.1,-21.2,5.7,-9.2;
move -80,-428.2,8,-21.2,5.8,-9.1;
move -81,-425.5,7.9,-21.2,5.9,-9.1;
move -81,-422.9,7.8,-21.2,6,-9.1;
move -82,-420.3,7.7,-21.6,6.2,-9;
move -82,-417.7,7.5,-21.6,6.3,-9;
move -83,-415.2,7.4,-21.6,6.4,-9;
move -83,-412.6,7.3,-21.6,6.5,-8.9;
move -83,-410.1,7.2,-21.6,6.6,-8.9;
move -83,-407.6,7,-21.6,6.7,-8.8;
move -83,-405.1,6.9,-21.6,6.8,-8.8;
move -83,-402.6,6.8,-21.6,6.9,-8.8;
move -83,-400.2,6.6,-21.6,7.1,-8.7;
move -83,-397.9,6.5,-21.6,7.2,-8.7;
move -83,-395.5,6.4,-21.6,7.3,-8.7;
move -83,-393.3,6.3,-21.6,7.4,-8.6;
move -82,-391,6.1,-21.6,7.5,-8.6;
move -82,-388.9,6,-21.2,7.6,-8.5;
move -82,-386.8,5.8,-21.2,7.7,-8.5;
move -81,-384.7,5.7,-21.6,7.8,-8.4;
move -81,-382.7,5.5,-21.6,7.9,-8.4;
move -80,-380.8,5.4,-21.2,8,-8.4;
move -80,-378.9,5.2,-21.2,8.1,-8.3;
move -79,-377.1,5.1,-21.2,8.2,-8.3;
move -78,-375.4,5,-20.8,8.3,-8.2;
move -78,-373.8,4.8,-20.8,8.4,-8.2;
move -77,-372.1,4.7,-20.4,8.5,-8.1;
move -76,-370.6,4.6,-20.4,8.7,-8.1;
move -76,-369.1,4.5,-20.4,8.8,-8;
move -75,-367.6,4.3,-20.4,8.9,-8;
move -74,-366.2,4.2,-20.4,9,-7.9;
move -74,-364.9,4.1,-20.4,9.1,-7.9;
move -73,-363.6,3.9,-20.4,9.2,-7.8;
move -73,-362.4,3.8,-20.4,9.3,-7.8;
move -72,-361.1,3.7,-20,9.4,-7.7;
move -71,-359.9,3.6,-20,9.4,-7.7;
move -70,-358.8,3.5,-20,9.5,-7.6;
move -69,-357.6,3.4,-19.6,9.6,-7.6;
move -69,-356.4,3.3,-19.2,9.7,-7.5;
move -68,-355.3,3.1,-19.2,9.8,-7.5;
move -67,-354.1,3,-19.2,9.9,-7.4;
move -67,-353,3,-19.2,10,-7.4;
move -66,-351.9,2.9,-19.2,10.1,-7.3;
move -66,-350.7,2.8,-19.2,10.2,-7.3;
move -66,-349.6,2.7,-19.6,10.3,-7.2;
move -65,-348.4,2.6,-19.2,10.4,-7.1;
move -65,-347.3,2.6,-19.2,10.5,-7.1;
move -64,-346.2,2.5,-19.2,10.6,-7;
move -63,-345.1,2.5,-18.8,10.7,-7;
move -62,-344,2.4,-18.8,10.7,-6.9;
move -61,-342.9,2.4,-18.8,10.8,-6.8;
move -60,-341.8,2.3,-18.4,10.9,-6.8;
move -59,-340.8,2.3,-18.4,11,-6.7;
move -58,-339.7,2.3,-18,11.1,-6.7;
move -57,-338.7,2.2,-18,11.2,-6.6;
move -56,-337.6,2.2,-18,11.3,-6.5;
move -56,-336.6,2.2,-17.6,11.3,-6.5;
move -55,-335.5,2.2,-17.6,11.4,-6.4;
move -54,-334.5,2.2,-17.6,11.5,-6.4;
move -53,-333.4,2.2,-17.6,11.6,-6.3;
move -52,-332.3,2.2,-17.2,11.7,-6.2;
move -51,-331.1,2.2,-17.2,11.7,-6.2;
move -49,-329.8,2.2,-17.2,11.8,-6.1;
move -48,-328.5,2.2,-16.8,11.9,-6;
move -47,-327.1,2.3,-16.8,12,-6;
move -46,-325.5,2.3,-16.4,12,-5.9;
move -44,-323.9,2.3,-16.4,12.1,-5.8;
move -43,-322.3,2.4,-16,12.2,-5.8;
move -41,-320.6,2.4,-16,12.3,-5.7;
move -39,-318.8,2.4,-15.6,12.3,-5.6;
move -38,-316.8,2.5,-15.6,12.4,-5.6;
move -36,-314.6,2.5,-15.2,12.5,-5.5;
move -34,-312.4,2.5,-14.8,12.5,-5.4;
move -32,-310,2.6,-14.8,12.6,-5.4;
move -30,-307.5,2.7,-14.4,12.7,-5.3;
move -28,-305,2.7,-14,12.7,-5.2;
move -26,-302.4,2.8,-13.6,12.8,-5.1;
move -23,-299.8,2.8,-13.6,12.9,-5.1;
move -21,-297.1,2.9,-13.2,12.9,-5;
move -19,-294.3,3,-12.8,13,-4.9;
move -16,-291.6,3.1,-12.4,13.1,-4.9;
move -14,-288.7,3.2,-12.4,13.1,-4.8;
move -11,-285.9,3.3,-12,13.2,-4.7;
move -8,-283.2,3.3,-11.2,13.2,-4.6;
move -5,-280.4,3.4,-11.2,13.3,-4.6;
move -2,-277.7,3.5,-10.8,13.4,-4.5;
move 1,-275.1,3.6,-10.4,13.4,-4.4;
move 4,-272.6,3.7,-9.6,13.5,-4.3;
move 7,-270.5,3.8,-9.2,13.5,-4.3;
move 11,-268.6,3.9,-8.8,13.6,-4.2;
move 14,-267,4,-8.4,13.6,-4.1;
move 18,-265.4,4,-8,13.7,-4;
move 21,-263.9,4.1,-7.2,13.7,-4;
move 25,-262.4,4.2,-6.8,13.8,-3.9;
move 29,-261,4.3,-6.4,13.8,-3.8;
move 32,-259.7,4.5,-6,13.9,-3.7;
move 36,-258.5,4.6,-5.2,13.9,-3.7;
move 40,-257.4,4.7,-4.8,14,-3.6;
move 44,-256.4,4.8,-4.4,14,-3.5;
move 48,-255.4,4.9,-3.6,14.1,-3.4;
move 52,-254.6,5,-3.2,14.1,-3.4;
move 56,-253.8,5.2,-2.8,14.1,-3.3;
move 60,-253,5.3,-2,14.2,-3.2;
move 64,-252.2,5.4,-1.6,14.2,-3.1;
move 67,-251.4,5.6,-1.2,14.3,-3;
move 71,-250.5,5.7,-0.4,14.3,-3;
move 75,-249.6,5.8,0,14.3,-2.9;
move 79,-248.6,5.9,0.8,14.4,-2.8;
move 83,-247.6,6.1,1.2,14.4,-2.7;
move 86,-246.4,6.2,1.6,14.4,-2.6;
move 90,-245.2,6.3,2,14.5,-2.6;
move 93,-244,6.5,2.4,14.5,-2.5;
move 96,-242.7,6.6,2.8,14.5,-2.4;
move 99,-241.4,6.8,3.6,14.6,-2.3;
move 102,-240.1,6.9,4,14.6,-2.2;
move 105,-238.9,7,4,14.6,-2.2;
move 108,-237.8,7.1,4.4,14.7,-2.1;
move 110,-236.7,7.3,4.8,14.7,-2;
move 112,-235.7,7.4,5.2,14.7,-1.9;
move 115,-235,7.5,5.6,14.7,-1.8;
move 117,-234.6,7.7,6,14.8,-1.8;
move 119,-234.5,7.8,6,14.8,-1.7;
move 120,-234.6,7.9,6.4,14.8,-1.6;
move 122,-235,8,6.4,14.8,-1.5;
move 123,-235.6,8.1,6.8,14.8,-1.4;
move 124,-236.6,8.3,6.8,14.9,-1.4;
move 125,-237.8,8.4,6.8,14.9,-1.3;
move 125,-239.2,8.5,7.2,14.9,-1.2;
move 125,-241,8.6,7.2,14.9,-1.1;
move 125,-242.9,8.7,7.2,14.9,-1;
move 125,-245.1,8.8,6.8,14.9,-0.9;
move 124,-247.4,8.9,6.8,14.9,-0.9;
move 123,-249.7,9,6.8,15,-0.8;
move 122,-252.1,9.1,6.4,15,-0.7;
move 121,-254.6,9.2,6.4,15,-0.6;
move 119,-257,9.3,6,15,-0.5;
move 117,-259.4,9.3,6,15,-0.5;
move 116,-261.7,9.4,5.6,15,-0.4;
move 113,-263.7,9.5,5.2,15,-0.3;
move 111,-265.7,9.5,5.2,15,-0.2;
move 109,-267.6,9.6,4.8,15,-0.1;
move 106,-269.4,9.7,4.4,15,-0;
move 103,-271.3,9.8,4,15,0;
move 100,-273,9.9,3.6,15,0.1;
move 96,-274.7,9.9,3.2,15,0.2;
move 92,-276.2,10,2.4,15,0.3;
move 88,-277.5,10.1,2,15,0.4;
move 84,-278.7,10.1,1.2,15,0.5;
move 80,-279.6,10.1,0.8,15,0.5;
move 76,-280.4,10.2,0,15,0.6;
move 71,-281,10.2,-0.4,15,0.7;
move 67,-281.6,10.2,-1.2,15,0.8;
move 62,-282,10.3,-1.6,14.9,0.9;
move 57,-282.4,10.3,-2.4,14.9,1;
move 52,-282.6,10.3,-3.2,14.9,1;
move 47,-282.9,10.4,-4,14.9,1.1;
move 42,-283,10.4,-4.4,14.9,1.2;
move 37,-283.1,10.4,-5.2,14.9,1.3;
move 32,-283.2,10.4,-6,14.9,1.4;
move 26,-283.3,10.5,-6.8,14.8,1.4;
move 21,-283.4,10.5,-7.2,14.8,1.5;
move 16,-283.4,10.5,-8,14.8,1.6;
move 10,-283.4,10.5,-8.8,14.8,1.7;
move 5,-283.5,10.5,-9.6,14.8,1.8;
move -1,-283.6,10.5,-10.4,14.7,1.9;
move -7,-283.6,10.5,-11.2,14.7,1.9;
move -12,-283.6,10.5,-12,14.7,2;
move -18,-283.6,10.5,-12.8,14.7,2.1;
move -23,-283.5,10.5,-13.6,14.6,2.2;
move -29,-283.4,10.5,-14.4,14.6,2.3;
move -34,-283.2,10.5,-14.8,14.6,2.3;
move -39,-282.9,10.4,-15.6,14.6,2.4;
move -44,-282.6,10.4,-16.4,14.5,2.5;
move -48,-282.1,10.4,-17.2,14.5,2.6;
move -53,-281.4,10.3,-18,14.5,2.7;
move -57,-280.5,10.3,-18.4,14.4,2.7;
move -61,-279.4,10.2,-18.8,14.4,2.8;
move -64,-278.1,10.2,-19.2,14.4,2.9;
move -68,-276.4,10.1,-19.6,14.3,3;
move -71,-274.4,10.1,-20,14.3,3.1;
move -74,-272,10,-20.4,14.2,3.1;
move -77,-269.2,10,-21.2,14.2,3.2;
move -80,-266,9.9,-21.2,14.2,3.3;
move -82,-262.4,9.8,-21.6,14.1,3.4;
move -84,-258.2,9.8,-22,14.1,3.4;
move -86,-253.6,9.7,-22.4,14,3.5;
move -87,-248.5,9.7,-22.4,14,3.6;
move -89,-242.8,9.6,-22.8,13.9,3.7;
move -89,-236.6,9.6,-22.8,13.9,3.7;
move -90,-230,9.5,-22.8,13.8,3.8;
move -90,-222.9,9.4,-22.8,13.8,3.9;
move -90,-215.3,9.4,-22.8,13.8,4;
move -90,-207.4,9.3,-22.8,13.7,4;
move -89,-199,9.2,-22.4,13.6,4.1;
move -88,-190.3,9.2,-22.4,13.6,4.2;
move -87,-181.2,9.1,-22.4,13.5,4.3;
move -85,-171.7,9,-22,13.5,4.3;
move -83,-161.9,9,-22,13.4,4.4;
move -81,-151.9,8.9,-21.6,13.4,4.5;
move -78,-141.7,8.8,-21.2,13.3,4.6;
move -75,-131.4,8.8,-20.8,13.3,4.6;
move -72,-121,8.7,-20.4,13.2,4.7;
move -68,-110.5,8.7,-20,13.1,4.8;
move -64,-100.2,8.6,-19.6,13.1,4.9;
move -60,-89.9,8.5,-18.8,13,4.9;
move -55,-79.8,8.5,-18,13,5;
move -50,-70,8.4,-17.2,12.9,5.1;
move -44,-60.6,8.4,-16.4,12.8,5.1;
move -39,-51.7,8.3,-15.6,12.8,5.2;
move -33,-43.3,8.3,-14.8,12.7,5.3;
move -27,-35.5,8.2,-14,12.6,5.4;
move -21,-28.3,8.2,-13.2,12.6,5.4;
move -15,-21.8,8.2,-12.4,12.5,5.5;
move -8,-16.1,8.1,-11.2,12.4,5.6;
move -2,-11.2,8.1,-10.4,12.4,5.6;
move 4,-7.1,8.1,-9.6,12.3,5.7;
move 11,-4.1,8.1,-8.8,12.2,5.8;
move 17,-1.9,8.1,-8,12.1,5.8;
move 24,-0.8,8.1,-7.2,12.1,5.9;
move 30,-0.7,8.1,-6,12,6;
move 37,-1.6,8.1,-5.2,11.9,6;
move 43,-3.7,8.1,-4.4,11.8,6.1;
move 49,-6.8,8.1,-3.2,11.8,6.2;
move 55,-11,8.1,-2.4,11.7,6.2;
move 62,-16.3,8.1,-1.6,11.6,6.3;
move 67,-22.8,8.2,-0.8,11.5,6.4;
move 73,-30.4,8.2,-0,11.4,6.4;
move 79,-39,8.2,0.4,11.4,6.5;
move 84,-48.6,8.3,1.2,11.3,6.6;
move 89,-59.1,8.3,2,11.2,6.6;
move 94,-70.4,8.3,2.8,11.1,6.7;
move 99,-82.4,8.4,3.6,11,6.7;
move 103,-95.1,8.4,4.4,10.9,6.8;
move 107,-108.3,8.5,4.8,10.9,6.9;
move 111,-122,8.5,5.2,10.8,6.9;
move 114,-135.9,8.6,5.6,10.7,7;
move 117,-150.1,8.6,6,10.6,7;
move 119,-164.4,8.7,6.4,10.5,7.1;
move 122,-178.8,8.7,6.8,10.4,7.2;
move 123,-193.1,8.8,6.8,10.3,7.2;
move 125,-207.3,8.8,7.2,10.2,7.3;
move 126,-221.3,8.9,7.2,10.1,7.3;
move 126,-235,8.9,7.2,10.1,7.4;
move 126,-248.3,8.9,7.2,10,7.4;
move 126,-261.2,9,7.2,9.9,7.5;
move 126,-273.6,9,7.2,9.8,7.5;
move 125,-285.4,9,7.2,9.7,7.6;
move 124,-296.7,9,7.2,9.6,7.7;
move 122,-307.3,9,6.8,9.5,7.7;
move 120,-317.1,9,6.4,9.4,7.8;
move 118,-326.1,9,6,9.3,7.8;
move 115,-334.3,9,5.6,9.2,7.9;
move 113,-341.6,9,5.2,9.1,7.9;
move 109,-347.9,9,4.8,9,8;
move 106,-353.3,9,4.4,8.9,8;
move 103,-357.6,9,4,8.8,8.1;
move 99,-360.9,8.9,3.2,8.7,8.1;
move 95,-363,8.9,2.8,8.6,8.1;
move 92,-364.1,8.8,2.4,8.5,8.2;
move 88,-364,8.8,1.6,8.4,8.2;
move 84,-363,8.7,1.2,8.3,8.3;
move 80,-360.9,8.7,0.4,8.2,8.3;
move 76,-357.9,8.6,0,8.1,8.4;
move 72,-353.9,8.6,-0.4,8,8.4;
move 68,-348.9,8.5,-1.2,7.9,8.5;
move 64,-343.1,8.4,-1.6,7.7,8.5;
move 60,-336.5,8.3,-2,7.6,8.5;
move 56,-329,8.2,-2.8,7.5,8.6;
move 52,-320.9,8.1,-3.2,7.4,8.6;
move 49,-312.2,8,-3.6,7.3,8.7;
move 45,-303.1,7.9,-4.4,7.2,8.7;
move 42,-293.6,7.8,-4.8,7.1,8.7;
move 39,-283.7,7.7,-5.2,7,8.8;
move 36,-273.5,7.5,-5.6,6.9,8.8;
move 33,-263,7.4,-6,6.8,8.9;
move 31,-252.2,7.2,-6.4,6.7,8.9;
move 29,-241.2,7.1,-6.4,6.5,8.9;
move 27,-230.1,6.9,-6.8,6.4,9;
move 25,-218.8,6.8,-7.2,6.3,9;
move 24,-207.3,6.6,-7.2,6.2,9;
move 23,-195.8,6.4,-7.6,6.1,9.1;
move 22,-184.2,6.2,-7.6,6,9.1;
move 21,-172.6,6,-7.6,5.9,9.2;
move 21,-160.9,5.8,-7.6,5.7,9.2;
move 20,-149.3,5.6,-7.6,5.6,9.2;
move 20,-137.7,5.4,-7.6,5.5,9.3;
move 20,-126.2,5.2,-7.6,5.4,9.3;
move 21,-114.9,5,-7.6,5.3,9.3;
move 21,-103.8,4.8,-7.6,5.2,9.4;
move 22,-93,4.6,-7.6,5,9.4;
move 23,-82.5,4.4,-7.6,4.9,9.4;
move 25,-72.4,4.2,-7.2,4.8,9.4;
move 26,-62.9,3.9,-6.8,4.7,9.5;
move 28,-54,3.7,-6.8,4.6,9.5;
move 30,-45.7,3.5,-6.4,4.4,9.5;
move 33,-38.2,3.2,-6,4.3,9.6;
move 36,-31.5,3,-5.6,4.2,9.6;
move 39,-25.5,2.8,-5.2,4.1,9.6;
move 42,-20.3,2.6,-4.8,4,9.6;
move 46,-15.9,2.4,-4.4,3.8,9.7;
move 49,-12.3,2.2,-3.6,3.7,9.7;
move 53,-9.4,2,-3.2,3.6,9.7;
move 58,-7.3,1.9,-2.4,3.5,9.7;
move 62,-5.8,1.7,-2,3.4,9.8;
move 66,-5,1.5,-1.2,3.2,9.8;
move 71,-4.8,1.3,-0.8,3.1,9.8;
move 76,-5,1.1,0,3,9.8;
move 81,-5.8,0.9,0.8,2.9,9.8;
move 86,-6.9,0.7,1.2,2.8,9.9;
move 90,-8.3,0.6,2,2.6,9.9;
move 96,-10,0.4,2.8,2.5,9.9;
move 101,-12,0.3,3.6,2.4,9.9;
move 106,-14.1,0.1,4,2.3,9.9;
move 111,-16.3,-0,4.8,2.1,9.9;
move 116,-18.7,-0.2,5.6,2,9.9;
move 121,-21.1,-0.3,6.4,1.9,9.9;
move 126,-23.6,-0.4,6.8,1.8,9.9;
move 131,-26.2,-0.5,7.6,1.6,9.9;
move 136,-28.8,-0.6,8.4,1.5,10;
move 140,-31.2,-0.7,8.8,1.4,10;
move 145,-33.7,-0.8,9.6,1.3,10;
move 150,-36.1,-0.9,10.4,1.1,10;
move 154,-38.6,-1,10.8,1,10;
move 159,-41,-1,11.6,0.9,10;
move 163,-43.6,-1.1,12,0.8,10;
move 167,-46.1,-1.2,12.4,0.6,10;
move 171,-48.8,-1.2,13.2,0.5,10;
move 175,-51.5,-1.3,13.6,0.4,10;
move 179,-54.3,-1.3,14.4,0.3,10;
move 183,-57.2,-1.3,14.8,0.1,10;
move 187,-60.1,-1.3,15.2,0,10;
move 190,-63.2,-1.3,15.6,0,10;
move 194,-66.3,-1.3,16.4,0,10;
move 197,-69.5,-1.3,16.8,0,10;
move 201,-72.9,-1.3,17.2,0,10;
move 204,-76.3,-1.3,17.6,0,10;
move 207,-79.8,-1.3,18,0,10;
move 210,-83.3,-1.3,18.4,0,10;
move 213,-86.9,-1.2,18.8,0,10;
move 216,-90.5,-1.2,19.2,0,10;
move 219,-94.1,-1.2,19.6,0,10;
move 221,-97.7,-1.1,20,0,10;
move 224,-101.3,-1.1,20.4,0,10;
move 226,-104.8,-1,20.8,0,9.9;
move 228,-108.2,-0.9,20.8,0,9.9;
move 230,-111.4,-0.9,21.2,0,9.9;
move 232,-114.5,-0.8,21.6,0,9.9;
move 234,-117.3,-0.7,21.6,0,9.9;
move 235,-120,-0.6,22,0,9.9;
move 237,-122.4,-0.6,22,0,9.9;
move 238,-124.6,-0.5,22.4,0,9.9;
move 239,-126.5,-0.4,22.4,0,9.9;
move 240,-128.1,-0.3,22.4,0,9.8;
move 241,-129.5,-0.2,22.8,0,9.8;
move 242,-130.6,-0.1,22.8,0,9.8;
move 243,-131.4,-0,22.8,0,9.8;
move 244,-131.9,0.1,22.8,0,9.8;
move 245,-132.1,0.2,22.8,0,9.7;
move 245,-132,0.3,23.2,0,9.7;
move 246,-131.7,0.4,23.2,0,9.7;
move 247,-131.2,0.5,23.2,0,9.7;
move 248,-130.5,0.6,23.6,0,9.7;
move 249,-129.7,0.7,23.6,0,9.6;
move 249,-128.8,0.8,23.6,0,9.6;
move 250,-127.8,0.9,24,0,9.6;
move 251,-126.9,1,24,0,9.5;
move 251,-126,1.1,24,0,9.5;
move 252,-125.3,1.2,24,0,9.5;
move 252,-124.7,1.3,24,0,9.5;
move 252,-124.3,1.4,24,0,9.4;
move 253,-124.3,1.6,24.4,0,9.4;
move 253,-124.5,1.7,24.4,0,9.4;
move 253,-125,1.8,24,0,9.3;
move 253,-125.9,1.9,24,0,9.3;
move 254,-127.2,2.1,24.4,0,9.3;
move 254,-128.8,2.2,24.4,0,9.2;
move 254,-130.8,2.3,24.4,0,9.2;
move 254,-133.2,2.4,24.4,0,9.2;
move 253,-135.9,2.5,24.4,0,9.1;
move 253,-138.9,2.7,24.4,0,9.1;
move 253,-142.1,2.8,24,0,9.1;
move 253,-145.6,2.9,24,0,9;
move 252,-149.2,3,24,0,9;
move 252,-153,3.1,24,0,9;
move 251,-156.9,3.2,24,0,8.9;
move 251,-160.8,3.3,24,0,8.9;
move 250,-164.8,3.4,24,0,8.8;
move 250,-168.8,3.5,23.6,0,8.8;
move 249,-172.8,3.6,23.6,0,8.8;
move 249,-176.7,3.8,23.6,0,8.7;
move 248,-180.6,3.9,23.6,0,8.7;
move 247,-184.4,4,23.6,0,8.7;
move 246,-188.2,4.1,23.2,0,8.6;
move 245,-191.9,4.2,23.2,0,8.6;
move 244,-195.6,4.3,23.2,0,8.5;
move 243,-199.2,4.4,22.8,0,8.5;
move 241,-202.8,4.5,22.4,0,8.4;
move 240,-206.4,4.7,22.4,0,8.4;
move 239,-209.9,4.7,22.4,0,8.4;
move 237,-213.5,4.8,22,0,8.3;
move 235,-217,4.9,22,0,8.3;
move 234,-220.5,5,21.6,0,8.2;
move 232,-223.9,5.1,21.6,0,8.2;
move 230,-227.3,5.1,21.2,0,8.1;
move 227,-230.6,5.2,20.8,0,8.1;
move 225,-233.9,5.3,20.4,0,8;
move 222,-237.2,5.4,20,0,8;
move 220,-240.5,5.5,19.6,0,7.9;
move 217,-243.7,5.5,19.2,0,7.9;
move 214,-246.8,5.6,18.8,0,7.8;
move 212,-249.8,5.7,18.8,0,7.8;
move 209,-252.8,5.8,18.4,0,7.7;
move 205,-255.7,5.8,18,0,7.7;
move 202,-258.6,5.9,17.2,0,7.6;
move 199,-261.3,6,16.8,0,7.6;
move 196,-263.9,6,16.4,0,7.5;
move 192,-266.4,6.1,16,0,7.5;
move 189,-268.8,6.1,15.6,0,7.4;
move 185,-271,6.2,14.8,-10,7.4;
move 181,-273.1,6.2,14.4,-10.1,7.3;
move 177,-275.1,6.3,14,-10.2,7.3;
move 174,-277,6.4,13.2,-10.3,7.2;
move 170,-278.7,6.4,12.8,-10.4,7.1;
move 166,-280.3,6.5,12.4,-10.5,7.1;
move 162,-281.7,6.5,11.6,-10.6,7;
move 158,-282.9,6.6,11.2,-10.7,7;
move 155,-283.9,6.6,10.8,-10.8,6.9;
move 151,-284.7,6.7,10.4,-10.8,6.8;
move 147,-285.3,6.7,9.6,-10.9,6.8;
move 144,-285.7,6.8,9.2,-11,6.7;
move 140,-286,6.9,8.8,-11.1,6.7;
move 137,-286.1,6.9,8.4,-11.2,6.6;
move 133,-285.9,7,8,-11.3,6.5;
move 130,-285.6,7.1,7.2,-11.3,6.5;
move 127,-285,7.1,6.8,-11.4,6.4;
move 124,-284.2,7.2,6.4,-11.5,6.4;
move 120,-283.2,7.3,6,-11.6,6.3;
move 117,-282,7.3,5.6,-11.7,6.2;
move 115,-280.7,7.4,5.2,-11.7,6.2;
move 112,-279.1,7.4,4.8,-11.8,6.1;
move 109,-277.3,7.5,4.4,-11.9,6;
move 107,-275.4,7.5,4,-12,6;
move 105,-273.3,7.6,4,-12,5.9;
move 102,-271,7.6,3.6,-12.1,5.8;
move 100,-268.7,7.6,3.2,-12.2,5.8;
move 98,-266.3,7.7,3.2,-12.3,5.7;
move 96,-263.9,7.7,2.8,-12.3,5.6;
move 94,-261.4,7.8,2.4,-12.4,5.6;
move 92,-258.9,7.8,2.4,-12.5,5.5;
move 90,-256.5,7.8,2,-12.5,5.4;
move 88,-254.1,7.8,1.6,-12.6,5.4;
move 86,-251.7,7.9,1.2,-12.7,5.3;
move 84,-249.4,7.9,1.2,-12.7,5.2;
move 83,-247.3,7.9,0.8,-12.8,5.1;
move 81,-245.2,7.9,0.8,-12.9,5.1;
move 80,-243.2,7.9,0.4,-12.9,5;
move 79,-241.4,7.9,0.4,-13,4.9;
move 78,-239.7,8,0,-13.1,4.9;
move 77,-238.1,8,-0,-13.1,4.8;
move 76,-236.7,8,-0,-13.2,4.7;
move 75,-235.4,8,-0.4,-13.2,4.6;
move 74,-234.2,8,-0,-13.3,4.6;
move 74,-233.3,8.1,-0.4,-13.4,4.5;
move 74,-232.5,8.1,-0.4,-13.4,4.4;
move 73,-231.9,8.1,-0.4,-13.5,4.3;
move 73,-231.4,8.2,-0.4,-13.5,4.3;
move 73,-231.1,8.2,-0.4,-13.6,4.2;
move 73,-231,8.2,-0.4,-13.6,4.1;
move 74,-231,8.2,-0.4,-13.7,4;
move 74,-231.2,8.1,-0.4,-13.7,4;
move 74,-231.5,8.2,-0,-13.8,3.9;
move 75,-231.9,8.1,-0,-13.8,3.8;
move 75,-232.5,8.1,0,-13.9,3.7;
move 75,-233.2,8.1,0,-13.9,3.7;
move 76,-234,8.1,0,-14,3.6;
move 76,-234.8,8.1,0,-14,3.5;
move 77,-235.7,8.1,0,-14.1,3.4;
move 77,-236.7,8,0.4,-14.1,3.3;
move 78,-237.6,8,0.4,-14.2,3.3;
move 78,-238.6,8,0.4,-14.2,3.2;
move 79,-239.5,8,0.4,-14.2,3.1;
move 79,-240.3,8,0.4,-14.3,3;
move 80,-241.2,7.9,0.4,-14.3,2.9;
move 80,-241.9,7.9,0.8,-14.3,2.9;
move 81,-242.6,7.9,0.8,-14.4,2.8;
move 82,-243.2,7.9,0.8,-14.4,2.7;
move 82,-243.8,7.8,0.8,-14.5,2.6;
move 83,-244.2,7.8,1.2,-14.5,2.5;
move 83,-244.6,7.8,1.2,-14.5,2.5;
move 84,-244.9,7.7,1.2,-14.5,2.4;
move 84,-245.1,7.7,1.2,-14.6,2.3;
move 85,-245.2,7.7,1.2,-14.6,2.2;
move 85,-245.3,7.6,1.2,-14.6,2.1;
move 86,-245.3,7.6,1.6,-14.7,2.1;
move 86,-245.3,7.5,1.6,-14.7,2;
move 86,-245.3,7.5,1.6,-14.7,1.9;
move 87,-245.3,7.4,1.6,-14.7,1.8;
move 87,-245.3,7.4,1.6,-14.8,1.7;
move 87,-245.4,7.3,1.6,-14.8,1.7;
move 87,-245.4,7.3,1.6,-14.8,1.6;
move 87,-245.6,7.2,1.6,-14.8,1.5;
move 87,-245.7,7.2,1.6,-14.8,1.4;
move 87,-245.9,7.1,1.6,-14.9,1.3;
move 87,-246.2,7.1,1.6,-14.9,1.2;
move 87,-246.5,7,1.6,-14.9,1.2;
move 87,-246.9,7,1.6,-14.9,1.1;
move 87,-247.4,6.9,1.6,-14.9,1;
move 87,-247.9,6.8,1.6,-14.9,0.9;
move 87,-248.4,6.8,1.6,-14.9,0.8;
move 87,-248.9,6.7,1.6,-15,0.8;
move 87,-249.5,6.7,1.6,-15,0.7;
move 87,-250,6.6,1.6,-15,0.6;
move 87,-250.6,6.5,1.6,-15,0.5;
move 87,-251.2,6.4,1.6,-15,0.4;
move 87,-251.9,6.4,1.6,-15,0.4;
move 87,-252.5,6.3,1.6,-15,0.3;
move 86,-253,6.2,1.6,-15,0.2;
move 86,-253.6,6.2,1.6,-15,0.1;
move 86,-254.1,6.1,1.6,-15,0;
move 85,-254.6,6,1.2,-15,-0.1;
move 85,-255,6,1.2,-15,-0.1;
move 84,-255.4,5.9,1.2,-15,-0.2;
move 84,-255.8,5.8,1.2,-15,-0.3;
move 83,-256.1,5.7,1.2,-15,-0.4;
move 83,-256.3,5.6,1.2,-15,-0.5;
move 82,-256.5,5.5,0.8,-15,-0.5;
move 81,-256.7,5.5,0.8,-15,-0.6;
move 81,-256.7,5.4,0.8,-15,-0.7;
move 80,-256.7,5.3,0.8,-15,-0.8;
move 79,-256.6,5.2,0.4,-14.9,-0.9;
move 79,-256.4,5.1,0.4,-14.9,-1;
move 78,-256.2,5,0.4,-14.9,-1;
move 78,-255.9,4.9,0.4,-14.9,-1.1;
move 77,-255.5,4.8,0,-14.9,-1.2;
move 77,-255,4.7,0,-14.9,-1.3;
move 76,-254.5,4.6,0,-14.9,-1.4;
move 76,-254,4.6,-0,-14.8,-1.5;
move 75,-253.4,4.5,-0,-14.8,-1.5;
move 75,-252.8,4.4,-0,-14.8,-1.6;
move 74,-252.1,4.3,-0,-14.8,-1.7;
move 74,-251.5,4.2,-0,-14.8,-1.8;
move 74,-250.9,4.1,-0.4,-14.7,-1.9;
move 73,-250.2,4,-0.4,-14.7,-1.9;
move 73,-249.6,3.9,-0.4,-14.7,-2;
move 72,-249,3.8,-0.4,-14.7,-2.1;
move 72,-248.5,3.7,-0.4,-14.6,-2.2;
move 71,-248,3.6,-0.4,-14.6,-2.3;
move 71,-247.5,3.5,-0.8,-14.6,-2.4;
move 70,-247.1,3.4,-0.8,-14.6,-2.4;
move 70,-246.7,3.4,-0.8,-14.5,-2.5;
move 69,-246.4,3.3,-0.8,-14.5,-2.6;
move 69,-246.2,3.2,-0.8,-14.5,-2.7;
move 68,-245.9,3.1,-0.8,-14.4,-2.8;
move 68,-245.7,3,-1.2,-14.4,-2.8;
move 68,-245.6,2.9,-1.2,-14.4,-2.9;
move 67,-245.4,2.8,-1.2,-14.3,-3;
move 67,-245.3,2.7,-1.2,-14.3,-3.1;
move 67,-245.3,2.6,-1.2,-14.2,-3.2;
move 67,-245.3,2.5,-1.2,-14.2,-3.2;
move 67,-245.3,2.4,-1.2,-14.2,-3.3;
move 67,-245.3,2.3,-1.2,-14.1,-3.4;
move 67,-245.3,2.2,-1.2,-14.1,-3.5;
move 67,-245.4,2.1,-1.2,-14,-3.5;
move 67,-245.4,2,-1.2,-14,-3.6;
move 67,-245.4,1.9,-1.2,-13.9,-3.7;
move 67,-245.4,1.8,-1.2,-13.9,-3.8;
move 67,-245.5,1.7,-1.2,-13.8,-3.9;
move 67,-245.5,1.6,-1.2,-13.8,-3.9;
move 68,-245.6,1.5,-1.2,-13.7,-4;
move 68,-245.7,1.4,-1.2,-13.7,-4.1;
move 68,-245.7,1.3,-0.8,-13.6,-4.2;
move 69,-245.7,1.2,-0.8,-13.6,-4.2;
move 69,-245.8,1.1,-0.8,-13.5,-4.3;
move 69,-245.8,1,-0.8,-13.5,-4.4;
move 70,-245.8,0.8,-0.8,-13.4,-4.5;
move 70,-245.8,0.7,-0.8,-13.4,-4.5;
move 70,-245.8,0.6,-0.8,-13.3,-4.6;
move 71,-245.7,0.5,-0.8,-13.3,-4.7;
move 71,-245.7,0.4,-0.4,-13.2,-4.8;
move 71,-245.7,0.2,-0.4,-13.1,-4.8;
move 72,-245.6,0.1,-0.4,-13.1,-4.9;
move 72,-245.5,0,-0.4,-13,-5;
move 73,-245.4,-0.1,-0.4,-13,-5;
move 73,-245.3,-0.3,-0.4,-12.9,-5.1;
move 74,-245.1,-0.4,-0.4,-12.8,-5.2;
move 74,-244.9,-0.5,-0.4,-12.8,-5.3;
move 75,-244.7,-0.6,-0,-12.7,-5.3;
move 76,-244.4,-0.8,-0,-12.6,-5.4;
move 77,-244.1,-0.9,0,-12.6,-5.5;
move 77,-243.7,-1,0.4,-12.5,-5.5;
move 78,-243.3,-1.2,0.4,-12.4,-5.6;
move 79,-242.8,-1.3,0.4,-12.3,-5.7;
move 80,-242.4,-1.5,0.8,-12.3,-5.7;
move 81,-241.8,-1.6,0.8,-12.2,-5.8;
move 82,-241.3,-1.8,0.8,-12.1,-5.9;
move 83,-240.7,-1.9,1.2,-12.1,-6;
move 84,-240.1,-2.1,1.2,-12,-6;
move 85,-239.5,-2.3,1.2,-11.9,-6.1;
move 85,-239,-2.4,1.2,-11.8,-6.1;
move 86,-238.4,-2.6,1.6,-11.8,-6.2;
move 87,-237.9,-2.7,1.6,-11.7,-6.3;
move 88,-237.4,-2.9,1.6,-11.6,-6.3;
move 89,-237,-3.1,2,-11.5,-6.4;
move 90,-236.6,-3.3,2,-11.4,-6.5;
move 91,-236.3,-3.4,2,-11.4,-6.5;
move 93,-236,-3.6,2.4,-11.3,-6.6;
move 94,-235.9,-3.8,2.4,-11.2,-6.7;
move 95,-235.8,-3.9,2.8,-11.1,-6.7;
move 96,-235.8,-4.1,2.8,-11,-6.8;
move 97,-235.9,-4.3,2.8,-10.9,-6.8;
move 98,-236.1,-4.5,3.2,-10.8,-6.9;
move 100,-236.4,-4.7,3.2,-10.8,-7;
move 101,-236.7,-4.8,3.6,-10.7,-7;
move 102,-237.1,-5,3.6,-10.6,-7.1;
move 103,-237.6,-5.2,4,-10.5,-7.1;
move 105,-238.1,-5.4,4,-10.4,-7.2;
move 106,-238.7,-5.6,4,-10.3,-7.2;
move 107,-239.3,-5.7,4.4,-10.2,-7.3;
move 108,-240,-5.9,4.4,-10.1,-7.4;
move 109,-240.7,-6,4.8,-10,-7.4;
move 110,-241.4,-6.2,4.8,-9.9,-7.5;
move 110,-242.1,-6.4,4.8,-9.9,-7.5;
move 111,-242.9,-6.5,4.8,-9.8,-7.6;
move 112,-243.6,-6.7,5.2,-9.7,-7.6;
move 113,-244.4,-6.8,5.2,-9.6,-7.7;
move 113,-245.2,-7,5.2,-9.5,-7.7;
move 114,-245.9,-7.1,5.2,-9.4,-7.8;
move 114,-246.7,-7.3,5.2,-9.3,-7.8;
move 115,-247.5,-7.4,5.2,-9.2,-7.9;
move 115,-248.4,-7.6,5.6,-9.1,-7.9;
move 116,-249.3,-7.8,5.6,-9,-8;
move 116,-250.2,-7.9,5.6,-8.9,-8;
move 117,-251.2,-8.1,5.6,-8.8,-8.1;
move 117,-252.2,-8.2,6,-8.7,-8.1;
move 117,-253.4,-8.3,6,-8.6,-8.2;
move 117,-254.5,-8.4,5.6,-8.5,-8.2;
move 117,-255.8,-8.6,6,-8.4,-8.3;
move 117,-257,-8.7,5.6,-8.3,-8.3;
move 117,-258.4,-8.8,5.6,-8.2,-8.4;
move 117,-259.7,-8.9,5.6,-8.1,-8.4;
move 117,-261.2,-9,5.6,-7.9,-8.4;
move 117,-262.6,-9.1,5.6,-7.8,-8.5;
move 116,-264,-9.1,5.6,-7.7,-8.5;
move 116,-265.5,-9.2,5.6,-7.6,-8.6;
move 116,-267,-9.3,5.6,-7.5,-8.6;
move 115,-268.5,-9.4,5.6,-7.4,-8.7;
move 115,-269.9,-9.4,5.6,-7.3,-8.7;
move 114,-271.3,-9.4,5.2,-7.2,-8.7;
move 113,-272.7,-9.5,5.2,-7.1,-8.8;
move 112,-274,-9.5,5.2,-7,-8.8;
move 111,-275.2,-9.5,4.8,-6.9,-8.8;
move 110,-276.3,-9.5,4.8,-6.7,-8.9;
move 109,-277.4,-9.5,4.8,-6.6,-8.9;
move 108,-278.4,-9.5,4.4,-6.5,-9;
move 107,-279.4,-9.5,4.4,-6.4,-9;
move 105,-280.3,-9.5,4,-6.3,-9;
move 104,-281.1,-9.5,4,-6.2,-9.1;
move 103,-281.8,-9.4,3.6,-6.1,-9.1;
move 101,-282.5,-9.4,3.6,-6,-9.1;
move 100,-283.1,-9.3,3.6,-5.8,-9.2;
move 98,-283.7,-9.3,3.2,-5.7,-9.2;
move 97,-284.2,-9.2,2.8,-5.6,-9.2;
move 95,-284.6,-9.1,2.8,-5.5,-9.3;
move 94,-285,-9,2.4,-5.4,-9.3;
move 92,-285.4,-8.9,2.4,-5.3,-9.3;
move 91,-285.7,-8.8,2,-5.1,-9.4;
move 89,-286,-8.7,2,-5,-9.4;
move 88,-286.2,-8.6,1.6,-4.9,-9.4;
move 86,-286.4,-8.4,1.6,-4.8,-9.5;
move 85,-286.5,-8.3,1.2,-4.7,-9.5;
move 83,-286.6,-8.1,1.2,-4.6,-9.5;
move 81,-286.6,-8,0.8,-4.4,-9.5;
move 79,-286.6,-7.8,0.4,-4.3,-9.6;
move 78,-286.5,-7.6,0.4,-4.2,-9.6;
move 76,-286.4,-7.5,0,-4.1,-9.6;
move 74,-286.3,-7.3,-0,-4,-9.7;
move 73,-286.1,-7.1,-0.4,-3.8,-9.7;
move 71,-285.8,-6.9,-0.8,-3.7,-9.7;
move 69,-285.6,-6.7,-0.8,-3.6,-9.7;
move 67,-285.2,-6.5,-1.2,-3.5,-9.7;
move 66,-284.9,-6.3,-1.2,-3.3,-9.8;
move 64,-284.5,-6.1,-1.6,-3.2,-9.8;
move 62,-284.1,-5.9,-1.6,-3.1,-9.8;
move 61,-283.7,-5.7,-2,-3,-9.8;
move 59,-283.2,-5.4,-2.4,-2.9,-9.8;
move 57,-282.8,-5.2,-2.4,-2.7,-9.9;
move 55,-282.3,-5,-2.8,-2.6,-9.9;
move 54,-281.7,-4.7,-2.8,-2.5,-9.9;
move 52,-281.2,-4.5,-3.2,-2.4,-9.9;
move 51,-280.6,-4.3,-3.6,-2.2,-9.9;
move 49,-280,-4,-3.6,-2.1,-9.9;
move 47,-279.4,-3.8,-4,-2,-9.9;
move 46,-278.7,-3.6,-4,-1.9,-9.9;
move 45,-278,-3.4,-4.4,-1.7,-9.9;
move 43,-277.3,-3.2,-4.4,-1.6,-9.9;
move 42,-276.6,-2.9,-4.4,-1.5,-10;
move 41,-275.9,-2.7,-4.8,-1.4,-10;
move 40,-275.1,-2.5,-4.8,-1.2,-10;
move 39,-274.4,-2.3,-5.2,-1.1,-10;
move 38,-273.7,-2.1,-5.2,-1,-10;
move 37,-273,-1.8,-5.2,-0.9,-10;
move 37,-272.3,-1.6,-5.2,-0.7,-10;
move 36,-271.5,-1.4,-5.2,-0.6,-10;
move 35,-270.8,-1.2,-5.6,-0.5,-10;
move 35,-270.1,-1,-5.6,-0.4,-10;
move 34,-269.3,-0.8,-5.6,-0.2,-10;
move 33,-268.6,-0.6,-5.6,-0.1,-10;
move 33,-267.8,-0.5,-6,0,-10;
move 32,-267.1,-0.3,-6,0.1,-10;
move 32,-266.4,-0.1,-6,0.3,-10;
move 32,-265.7,0.1,-6,0.4,-10;
move 31,-265,0.3,-6,0.5,-10;
move 31,-264.2,0.5,-6,0.6,-10;
move 31,-263.5,0.6,-6,0.8,-10;
move 31,-262.8,0.8,-6,0.9,-10;
move 30,-262,0.9,-6,1,-10;
move 30,-261.3,1.1,-6.4,1.1,-10;
move 30,-260.5,1.2,-6.4,1.3,-10;
move 30,-259.8,1.4,-6.4,1.4,-10;
move 30,-259.1,1.5,-6,1.5,-10;
move 30,-258.3,1.6,-6,1.6,-9.9;
move 31,-257.6,1.7,-6.4,1.7,-9.9;
move 31,-256.8,1.8,-6,1.9,-9.9;
move 31,-256.1,1.9,-6,2,-9.9;
move 32,-255.4,2,-6,2.1,-9.9;
move 32,-254.6,2.1,-6,2.2,-9.9;
move 32,-253.9,2.2,-6,2.4,-9.9;
move 33,-253.3,2.3,-5.6,2.5,-9.9;
move 34,-252.6,2.4,-5.6,2.6,-9.9;
move 34,-252,2.4,-5.6,2.7,-9.8;
move 35,-251.4,2.5,-5.6,2.9,-9.8;
move 35,-250.8,2.5,-5.6,3,-9.8;
move 36,-250.2,2.6,-5.6,3.1,-9.8;
move 37,-249.7,2.7,-5.2,3.2,-9.8;
move 38,-249.2,2.7,-5.2,3.3,-9.7;
move 39,-248.8,2.7,-4.8,3.5,-9.7;
move 39,-248.4,2.8,-4.8,3.6,-9.7;
move 40,-248,2.8,-4.8,3.7,-9.7;
move 41,-247.6,2.8,-4.8,3.8,-9.7;
move 42,-247.3,2.8,-4.4,4,-9.6;
move 43,-247,2.8,-4.4,4.1,-9.6;
move 44,-246.7,2.8,-4.4,4.2,-9.6;
move 45,-246.5,2.9,-4,4.3,-9.5;
move 46,-246.2,2.9,-4,4.4,-9.5;
move 47,-246,2.9,-4,4.6,-9.5;
move 48,-245.7,2.9,-3.6,4.7,-9.5;
move 49,-245.4,2.9,-3.6,4.8,-9.4;
move 51,-245.1,2.9,-3.2,4.9,-9.4;
move 52,-244.8,2.8,-3.2,5,-9.4;
move 53,-244.5,2.8,-3.2,5.1,-9.3;
move 54,-244.2,2.8,-2.8,5.3,-9.3;
move 55,-243.9,2.8,-2.8,5.4,-9.3;
move 57,-243.6,2.7,-2.4,5.5,-9.2;
move 58,-243.2,2.7,-2.4,5.6,-9.2;
move 59,-242.9,2.7,-2.4,5.7,-9.2;
move 60,-242.5,2.7,-2,5.8,-9.1;
move 61,-242.2,2.6,-2,6,-9.1;
move 63,-241.8,2.6,-1.6,6.1,-9.1;
move 64,-241.5,2.5,-1.6,6.2,-9;
move 65,-241.1,2.5,-1.2,6.3,-9;
move 66,-240.8,2.4,-1.2,6.4,-9;
move 67,-240.5,2.4,-1.2,6.5,-8.9;
move 69,-240.2,2.4,-0.8,6.6,-8.9;
move 70,-240,2.3,-0.8,6.8,-8.8;
move 71,-239.8,2.3,-0.8,6.9,-8.8;
move 72,-239.6,2.2,-0.4,7,-8.8;
move 73,-239.5,2.2,-0.4,7.1,-8.7;
move 75,-239.5,2.1,-0,7.2,-8.7;
move 76,-239.5,2.1,0,7.3,-8.7;
move 77,-239.5,2,0.4,7.4,-8.6;
move 79,-239.6,2,0.4,7.5,-8.6;
move 80,-239.8,2,0.8,7.6,-8.5;
